LIN {X 0,Y 144.549,Z 370.18,A -85,B 0,C 180,E1 -24511.717,E2 -24511.717} C_VEL
LIN {X 0,Y 147,Z 373.251,A -85,B 0,C 180,E1 -24513.717,E2 -24513.717} C_VEL
LIN {X 0,Y 149.193,Z 377.596,A -85,B 0,C 180,E1 -24515.66,E2 -24515.66} C_VEL
LIN {X 0,Y 150.4,Z 379.371,A -85,B 0,C 180,E1 -24516.571,E2 -24516.571} C_VEL
LIN {X 0,Y 153.159,Z 385.359,A -85,B 0,C 180,E1 -24519.038,E2 -24519.038} C_VEL
LIN {X 0,Y 155.845,Z 391.898,A -85,B 0,C 180,E1 -24521.494,E2 -24521.494} C_VEL
LIN {X 0,Y 158.018,Z 400.093,A -85,B 0,C 180,E1 -24524.224,E2 -24524.224} C_VEL
LIN {X 0,Y 159.382,Z 409.972,A -85,B 0,C 180,E1 -24527.295,E2 -24527.295} C_VEL
LIN {X 0,Y 159.68,Z 420.278,A -85,B 0,C 180,E1 -24530.574,E2 -24530.574} C_VEL
LIN {X 0,Y 159.24,Z 428.16,A -85,B 0,C 180,E1 -24533.244,E2 -24533.244} C_VEL
LIN {X 0,Y 158.452,Z 434.433,A -85,B 0,C 180,E1 -24535.562,E2 -24535.562} C_VEL
LIN {X 0,Y 157.349,Z 437.828,A -85,B 0,C 180,E1 -24536.829,E2 -24536.829} C_VEL
LIN {X 0,Y 154.356,Z 444.029,A -85,B 0,C 180,E1 -24539.188,E2 -24539.188} C_VEL
LIN {X 0,Y 151.022,Z 450.566,A -85,B 0,C 180,E1 -24542.266,E2 -24542.266} C_VEL
LIN {X 0,Y 148.76,Z 455.072,A -85,B 0,C 180,E1 -24544.837,E2 -24544.837} C_VEL
LIN {X 0,Y 145.707,Z 460.563,A -85,B 0,C 180,E1 -24548.792,E2 -24548.792} C_VEL
LIN {X 0,Y 143.312,Z 464.89,A -85,B 0,C 180,E1 -24552.888,E2 -24552.888} C_VEL
LIN {X 0,Y 142.247,Z 467.263,A -85,B 0,C 180,E1 -24555.698,E2 -24555.698} C_VEL
LIN {X 0,Y 141.417,Z 469.068,A -85,B 0,C 180,E1 -24558.534,E2 -24558.534} C_VEL
LIN {X 0,Y 140.617,Z 471.529,A -85,B 0,C 180,E1 -24564.263,E2 -24564.263} C_VEL
LIN {X 0,Y 140.572,Z 472.282,A -85,B 0,C 180,E1 -24569.356,E2 -24569.356} C_VEL
LIN {X 0,Y 140.49,Z 472.123,A -85,B 0,C 180,E1 -24572.867,E2 -24572.867} C_VEL
LIN {X 0,Y 140.558,Z 471.527,A -85,B 0,C 180,E1 -24575.739,E2 -24575.739} C_VEL
LIN {X 0,Y 141.417,Z 469.068,A -85,B 0,C 180,E1 -24581.466,E2 -24581.466} C_VEL
LIN {X 0,Y 142.743,Z 466.11,A -85,B 0,C 180,E1 -24585.712,E2 -24585.712} C_VEL
LIN {X 0,Y 144.851,Z 462.118,A -85,B 0,C 180,E1 -24589.854,E2 -24589.854} C_VEL
LIN {X 0,Y 147.632,Z 456.986,A -85,B 0,C 180,E1 -24593.869,E2 -24593.869} C_VEL
LIN {X 0,Y 150.506,Z 451.725,A -85,B 0,C 180,E1 -24597.083,E2 -24597.083} C_VEL
LIN {X 0,Y 153.633,Z 445.404,A -85,B 0,C 180,E1 -24600.212,E2 -24600.212} C_VEL
LIN {X 0,Y 156.52,Z 439.453,A -85,B 0,C 180,E1 -24602.603,E2 -24602.603} C_VEL
LIN {X 0,Y 158.012,Z 436.197,A -85,B 0,C 180,E1 -24603.777,E2 -24603.777} C_VEL
LIN {X 0,Y 159.052,Z 429.716,A -85,B 0,C 180,E1 -24606.175,E2 -24606.175} C_VEL
LIN {X 0,Y 159.597,Z 422.251,A -85,B 0,C 180,E1 -24608.752,E2 -24608.752} C_VEL
LIN {X 0,Y 159.582,Z 414.231,A -85,B 0,C 180,E1 -24611.345,E2 -24611.345} C_VEL
LIN {X 0,Y 158.977,Z 406.419,A -85,B 0,C 180,E1 -24613.776,E2 -24613.776} C_VEL
LIN {X 0,Y 157.376,Z 397.352,A -85,B 0,C 180,E1 -24616.635,E2 -24616.635} C_VEL
LIN {X 0,Y 154.927,Z 389.38,A -85,B 0,C 180,E1 -24619.399,E2 -24619.399} C_VEL
LIN {X 0,Y 152.629,Z 383.818,A -85,B 0,C 180,E1 -24621.516,E2 -24621.516} C_VEL
LIN {X 0,Y 150.401,Z 379.369,A -85,B 0,C 180,E1 -24623.429,E2 -24623.429} C_VEL
LIN {X 0,Y 147.643,Z 374.742,A -85,B 0,C 180,E1 -24625.66,E2 -24625.66} C_VEL
LIN {X 0,Y 147.013,Z 373.191,A -85,B 0,C 180,E1 -24626.286,E2 -24626.286} C_VEL
LIN {X 0,Y 144.636,Z 370.361,A -85,B 0,C 180,E1 -24628.202,E2 -24628.202} C_VEL
LIN {X 0,Y 143.643,Z 367.692,A -85,B 0,C 180,E1 -24629.188,E2 -24629.188} C_VEL
LIN {X 0,Y 143.541,Z 367.179,A -85,B 0,C 180,E1 -24629.469,E2 -24629.469} C_VEL
LIN {X 0,Y 143.504,Z 367.059,A -85,B 0,C 180,E1 -24629.933,E2 -24629.933} C_VEL
LIN {X 0,Y 142.747,Z 366.562,A -85,B 0,C 180,E1 -24632.267,E2 -24632.267} C_VEL
LIN {X 0,Y 141.148,Z 366.234,A -85,B 0,C 180,E1 -24634.575,E2 -24634.575} C_VEL
LIN {X 0,Y 136.612,Z 365.578,A -85,B 0,C 180,E1 -24640.934,E2 -24640.934} C_VEL
LIN {X 0,Y 136.249,Z 365.35,A -85,B 0,C 180,E1 -24642.612,E2 -24642.612} C_VEL
LIN {X 0,Y 136.498,Z 364.983,A -85,B 0,C 180,E1 -24648.113,E2 -24648.113} C_VEL
LIN {X 0,Y 136.59,Z 364.972,A -85,B 0,C 180,E1 -24651.119,E2 -24651.119} C_VEL
LIN {X 0,Y 137.133,Z 364.867,A -85,B 0,C 180,E1 -24659.998,E2 -24659.998} C_VEL
LIN {X 0,Y 136.588,Z 364.962,A -85,B 0,C 180,E1 -24668.878,E2 -24668.878} C_VEL
LIN {X 0,Y 136.491,Z 364.984,A -85,B 0,C 180,E1 -24671.953,E2 -24671.953} C_VEL
LIN {X 0,Y 136.243,Z 365.011,A -85,B 0,C 180,E1 -24678.028,E2 -24678.028} C_VEL
LIN {X 0,Y 136.195,Z 365.018,A -85,B 0,C 180,E1 -24681.745,E2 -24681.745} C_VEL
LIN {X 0,Y 136.072,Z 365.05,A -85,B 0,C 180,E1 -24685.117,E2 -24685.117} C_VEL
LIN {X 0,Y 136.885,Z 367.482,A -85,B 0,C 180,E1 -24686.283,E2 -24686.283} C_VEL
LIN {X 0,Y 139.006,Z 369.899,A -85,B 0,C 180,E1 -24688.562,E2 -24688.562} C_VEL
LIN {X 0,Y 140.078,Z 370.732,A -85,B 0,C 180,E1 -24689.546,E2 -24689.546} C_VEL
LIN {X 0,Y 141.571,Z 373.697,A -85,B 0,C 180,E1 -24691.206,E2 -24691.206} C_VEL
LIN {X 0,Y 143.657,Z 376.017,A -85,B 0,C 180,E1 -24693.014,E2 -24693.014} C_VEL
LIN {X 0,Y 145.288,Z 378.918,A -85,B 0,C 180,E1 -24694.681,E2 -24694.681} C_VEL
LIN {X 0,Y 146.643,Z 381.055,A -85,B 0,C 180,E1 -24695.949,E2 -24695.949} C_VEL
LIN {X 0,Y 150.21,Z 387.174,A -85,B 0,C 180,E1 -24699.196,E2 -24699.196} C_VEL
LIN {X 0,Y 154.208,Z 395.585,A -85,B 0,C 180,E1 -24703.125,E2 -24703.125} C_VEL
LIN {X 0,Y 157.583,Z 404.814,A -85,B 0,C 180,E1 -24707.071,E2 -24707.071} C_VEL
LIN {X 0,Y 159.742,Z 412.862,A -85,B 0,C 180,E1 -24710.371,E2 -24710.371} C_VEL
LIN {X 0,Y 161.215,Z 420.7,A -85,B 0,C 180,E1 -24713.626,E2 -24713.626} C_VEL
LIN {X 0,Y 162.339,Z 429.067,A -85,B 0,C 180,E1 -24717.358,E2 -24717.358} C_VEL
LIN {X 0,Y 164.398,Z 436.642,A -85,B 0,C 180,E1 -24721.38,E2 -24721.38} C_VEL
LIN {X 0,Y 167.404,Z 442.696,A -85,B 0,C 180,E1 -24725.177,E2 -24725.177} C_VEL
LIN {X 0,Y 172.404,Z 448.692,A -85,B 0,C 180,E1 -24729.647,E2 -24729.647} C_VEL
LIN {X 0,Y 176.708,Z 452.183,A -85,B 0,C 180,E1 -24732.65,E2 -24732.65} C_VEL
LIN {X 0,Y 183.948,Z 456.194,A -85,B 0,C 180,E1 -24736.748,E2 -24736.748} C_VEL
LIN {X 0,Y 192.327,Z 459.212,A -85,B 0,C 180,E1 -24740.613,E2 -24740.613} C_VEL
LIN {X 0,Y 200.809,Z 461.137,A -85,B 0,C 180,E1 -24743.973,E2 -24743.973} C_VEL
LIN {X 0,Y 206.606,Z 462.007,A -85,B 0,C 180,E1 -24746.099,E2 -24746.099} C_VEL
LIN {X 0,Y 211.968,Z 462.427,A -85,B 0,C 180,E1 -24748.1,E2 -24748.1} C_VEL
LIN {X 0,Y 216.26,Z 462.479,A -85,B 0,C 180,E1 -24750,E2 -24750} C_VEL
LIN {X 0,Y 211.001,Z 462.357,A -85,B 0,C 180,E1 -24752.268,E2 -24752.268} C_VEL
LIN {X 0,Y 204.488,Z 461.751,A -85,B 0,C 180,E1 -24754.674,E2 -24754.674} C_VEL
LIN {X 0,Y 195.012,Z 459.95,A -85,B 0,C 180,E1 -24758.288,E2 -24758.288} C_VEL
LIN {X 0,Y 186.73,Z 457.364,A -85,B 0,C 180,E1 -24761.89,E2 -24761.89} C_VEL
LIN {X 0,Y 178.969,Z 453.628,A -85,B 0,C 180,E1 -24765.955,E2 -24765.955} C_VEL
LIN {X 0,Y 174.544,Z 450.62,A -85,B 0,C 180,E1 -24768.791,E2 -24768.791} C_VEL
LIN {X 0,Y 169.212,Z 445.25,A -85,B 0,C 180,E1 -24773.038,E2 -24773.038} C_VEL
LIN {X 0,Y 165.598,Z 439.388,A -85,B 0,C 180,E1 -24776.974,E2 -24776.974} C_VEL
LIN {X 0,Y 163.29,Z 433.068,A -85,B 0,C 180,E1 -24780.596,E2 -24780.596} C_VEL
LIN {X 0,Y 161.752,Z 425.235,A -85,B 0,C 180,E1 -24784.391,E2 -24784.391} C_VEL
LIN {X 0,Y 160.923,Z 418.763,A -85,B 0,C 180,E1 -24787.157,E2 -24787.157} C_VEL
LIN {X 0,Y 159.111,Z 410.213,A -85,B 0,C 180,E1 -24790.681,E2 -24790.681} C_VEL
LIN {X 0,Y 156.632,Z 401.905,A -85,B 0,C 180,E1 -24794.12,E2 -24794.12} C_VEL
LIN {X 0,Y 152.879,Z 392.58,A -85,B 0,C 180,E1 -24798.199,E2 -24798.199} C_VEL
LIN {X 0,Y 148.813,Z 384.555,A -85,B 0,C 180,E1 -24802.126,E2 -24802.126} C_VEL
LIN {X 0,Y 145.995,Z 379.751,A -85,B 0,C 180,E1 -24804.716,E2 -24804.716} C_VEL
LIN {X 0,Y 143.91,Z 376.585,A -85,B 0,C 180,E1 -24806.707,E2 -24806.707} C_VEL
LIN {X 0,Y 143.077,Z 375.23,A -85,B 0,C 180,E1 -24807.505,E2 -24807.505} C_VEL
LIN {X 0,Y 140.821,Z 372.533,A -85,B 0,C 180,E1 -24809.546,E2 -24809.546} C_VEL
LIN {X 0,Y 139.937,Z 370.486,A -85,B 0,C 180,E1 -24810.609,E2 -24810.609} C_VEL
LIN {X 0,Y 137.39,Z 368.266,A -85,B 0,C 180,E1 -24813.105,E2 -24813.105} C_VEL
LIN {X 0,Y 136.236,Z 365.864,A -85,B 0,C 180,E1 -24814.609,E2 -24814.609} C_VEL
LIN {X 0,Y 136.075,Z 365.024,A -85,B 0,C 180,E1 -24814.986,E2 -24814.986} C_VEL
LIN {X 0,Y 136.24,Z 365.008,A -85,B 0,C 180,E1 -24818.834,E2 -24818.834} C_VEL
LIN {X 0,Y 136.275,Z 365,A -85,B 0,C 180,E1 -24825.059,E2 -24825.059} C_VEL
LIN {X 0,Y 136.497,Z 364.983,A -85,B 0,C 180,E1 -24828.116,E2 -24828.116} C_VEL
LIN {X 0,Y 136.588,Z 364.962,A -85,B 0,C 180,E1 -24831.122,E2 -24831.122} C_VEL
LIN {X 0,Y 137.133,Z 364.867,A -85,B 0,C 180,E1 -24840.002,E2 -24840.002} C_VEL
LIN {X 0,Y 136.59,Z 364.971,A -85,B 0,C 180,E1 -24848.881,E2 -24848.881} C_VEL
LIN {X 0,Y 136.492,Z 364.987,A -85,B 0,C 180,E1 -24851.956,E2 -24851.956} C_VEL
LIN {X 0,Y 136.266,Z 365.014,A -85,B 0,C 180,E1 -24854.946,E2 -24854.946} C_VEL
LIN {X 0,Y 136.365,Z 366.025,A -85,B 0,C 180,E1 -24861.149,E2 -24861.149} C_VEL
LIN {X 0,Y 136.373,Z 366.981,A -85,B 0,C 180,E1 -24865.163,E2 -24865.163} C_VEL
LIN {X 0,Y 137.366,Z 369.881,A -85,B 0,C 180,E1 -24866.494,E2 -24866.494} C_VEL
LIN {X 0,Y 139.889,Z 372.994,A -85,B 0,C 180,E1 -24869.09,E2 -24869.09} C_VEL
LIN {X 0,Y 140.452,Z 373.735,A -85,B 0,C 180,E1 -24869.645,E2 -24869.645} C_VEL
LIN {X 0,Y 141.954,Z 377.052,A -85,B 0,C 180,E1 -24871.324,E2 -24871.324} C_VEL
LIN {X 0,Y 143.821,Z 379.604,A -85,B 0,C 180,E1 -24872.975,E2 -24872.975} C_VEL
LIN {X 0,Y 144.834,Z 382.056,A -85,B 0,C 180,E1 -24874.089,E2 -24874.089} C_VEL
LIN {X 0,Y 146.097,Z 384.055,A -85,B 0,C 180,E1 -24875.26,E2 -24875.26} C_VEL
LIN {X 0,Y 149.265,Z 391.3,A -85,B 0,C 180,E1 -24878.473,E2 -24878.473} C_VEL
LIN {X 0,Y 151.684,Z 399.019,A -85,B 0,C 180,E1 -24881.508,E2 -24881.508} C_VEL
LIN {X 0,Y 152.964,Z 406.059,A -85,B 0,C 180,E1 -24883.989,E2 -24883.989} C_VEL
LIN {X 0,Y 153.587,Z 414.007,A -85,B 0,C 180,E1 -24886.656,E2 -24886.656} C_VEL
LIN {X 0,Y 153.528,Z 422.357,A -85,B 0,C 180,E1 -24889.526,E2 -24889.526} C_VEL
LIN {X 0,Y 152.845,Z 430.118,A -85,B 0,C 180,E1 -24892.368,E2 -24892.368} C_VEL
LIN {X 0,Y 151.94,Z 435.994,A -85,B 0,C 180,E1 -24894.677,E2 -24894.677} C_VEL
LIN {X 0,Y 150.614,Z 439.258,A -85,B 0,C 180,E1 -24895.948,E2 -24895.948} C_VEL
LIN {X 0,Y 147.524,Z 445.208,A -85,B 0,C 180,E1 -24898.397,E2 -24898.397} C_VEL
LIN {X 0,Y 144.204,Z 451.389,A -85,B 0,C 180,E1 -24901.535,E2 -24901.535} C_VEL
LIN {X 0,Y 142.365,Z 454.876,A -85,B 0,C 180,E1 -24903.622,E2 -24903.622} C_VEL
LIN {X 0,Y 139.085,Z 460.367,A -85,B 0,C 180,E1 -24907.73,E2 -24907.73} C_VEL
LIN {X 0,Y 136.507,Z 464.693,A -85,B 0,C 180,E1 -24912.007,E2 -24912.007} C_VEL
LIN {X 0,Y 135.35,Z 467.067,A -85,B 0,C 180,E1 -24914.952,E2 -24914.952} C_VEL
LIN {X 0,Y 134.451,Z 468.872,A -85,B 0,C 180,E1 -24917.931,E2 -24917.931} C_VEL
LIN {X 0,Y 133.543,Z 471.333,A -85,B 0,C 180,E1 -24923.958,E2 -24923.958} C_VEL
LIN {X 0,Y 133.414,Z 471.927,A -85,B 0,C 180,E1 -24926.98,E2 -24926.98} C_VEL
LIN {X 0,Y 133.535,Z 472.088,A -85,B 0,C 180,E1 -24930,E2 -24930} C_VEL
LIN {X 0,Y 133.401,Z 471.927,A -85,B 0,C 180,E1 -24933.02,E2 -24933.02} C_VEL
LIN {X 0,Y 133.474,Z 471.331,A -85,B 0,C 180,E1 -24936.045,E2 -24936.045} C_VEL
LIN {X 0,Y 134.451,Z 468.872,A -85,B 0,C 180,E1 -24942.069,E2 -24942.069} C_VEL
LIN {X 0,Y 135.882,Z 465.913,A -85,B 0,C 180,E1 -24946.527,E2 -24946.527} C_VEL
LIN {X 0,Y 138.157,Z 461.921,A -85,B 0,C 180,E1 -24950.86,E2 -24950.86} C_VEL
LIN {X 0,Y 141.146,Z 456.79,A -85,B 0,C 180,E1 -24955.039,E2 -24955.039} C_VEL
LIN {X 0,Y 143.579,Z 452.685,A -85,B 0,C 180,E1 -24957.711,E2 -24957.711} C_VEL
LIN {X 0,Y 146.722,Z 446.721,A -85,B 0,C 180,E1 -24960.912,E2 -24960.912} C_VEL
LIN {X 0,Y 149.771,Z 440.883,A -85,B 0,C 180,E1 -24963.461,E2 -24963.461} C_VEL
LIN {X 0,Y 151.95,Z 435.994,A -85,B 0,C 180,E1 -24965.32,E2 -24965.32} C_VEL
LIN {X 0,Y 153.22,Z 427.209,A -85,B 0,C 180,E1 -24968.759,E2 -24968.759} C_VEL
LIN {X 0,Y 153.66,Z 417.036,A -85,B 0,C 180,E1 -24972.333,E2 -24972.333} C_VEL
LIN {X 0,Y 153.18,Z 408.386,A -85,B 0,C 180,E1 -24975.269,E2 -24975.269} C_VEL
LIN {X 0,Y 152.083,Z 400.634,A -85,B 0,C 180,E1 -24977.924,E2 -24977.924} C_VEL
LIN {X 0,Y 149.973,Z 393.209,A -85,B 0,C 180,E1 -24980.705,E2 -24980.705} C_VEL
LIN {X 0,Y 147.368,Z 387.012,A -85,B 0,C 180,E1 -24983.405,E2 -24983.405} C_VEL
LIN {X 0,Y 145.745,Z 383.501,A -85,B 0,C 180,E1 -24985.06,E2 -24985.06} C_VEL
LIN {X 0,Y 143.906,Z 379.83,A -85,B 0,C 180,E1 -24986.932,E2 -24986.932} C_VEL
LIN {X 0,Y 143.251,Z 378.671,A -85,B 0,C 180,E1 -24987.546,E2 -24987.546} C_VEL
LIN {X 0,Y 141.051,Z 375.424,A -85,B 0,C 180,E1 -24989.598,E2 -24989.598} C_VEL
LIN {X 0,Y 140.309,Z 373.275,A -85,B 0,C 180,E1 -24990.551,E2 -24990.551} C_VEL
LIN {X 0,Y 137.672,Z 370.389,A -85,B 0,C 180,E1 -24993.161,E2 -24993.161} C_VEL
LIN {X 0,Y 136.526,Z 367.751,A -85,B 0,C 180,E1 -24994.562,E2 -24994.562} C_VEL
LIN {X 0,Y 136.352,Z 366.837,A -85,B 0,C 180,E1 -24995.037,E2 -24995.037} C_VEL
LIN {X 0,Y 136.365,Z 366.023,A -85,B 0,C 180,E1 -24998.851,E2 -24998.851} C_VEL
LIN {X 0,Y 136.249,Z 365.35,A -85,B 0,C 180,E1 -25002.612,E2 -25002.612} C_VEL
LIN {X 0,Y 135.519,Z 365.197,A -85,B 0,C 180,E1 -25005.082,E2 -25005.082} C_VEL
LIN {X 0,Y 133.954,Z 365.311,A -85,B 0,C 180,E1 -25007.524,E2 -25007.524} C_VEL
LIN {X 0,Y 129.763,Z 365.821,A -85,B 0,C 180,E1 -25014.266,E2 -25014.266} C_VEL
LIN {X 0,Y 129.594,Z 365.838,A -85,B 0,C 180,E1 -25016.037,E2 -25016.037} C_VEL
LIN {X 0,Y 130.089,Z 365.742,A -85,B 0,C 180,E1 -25019.998,E2 -25019.998} C_VEL
LIN {X 0,Y 129.514,Z 365.841,A -85,B 0,C 180,E1 -25029.367,E2 -25029.367} C_VEL
LIN {X 0,Y 129.392,Z 365.867,A -85,B 0,C 180,E1 -25032.546,E2 -25032.546} C_VEL
LIN {X 0,Y 129.195,Z 365.966,A -85,B 0,C 180,E1 -25037.611,E2 -25037.611} C_VEL
LIN {X 0,Y 129.963,Z 368.398,A -85,B 0,C 180,E1 -25039.341,E2 -25039.341} C_VEL
LIN {X 0,Y 132.558,Z 371.16,A -85,B 0,C 180,E1 -25043.164,E2 -25043.164} C_VEL
LIN {X 0,Y 133.403,Z 371.849,A -85,B 0,C 180,E1 -25044.199,E2 -25044.199} C_VEL
LIN {X 0,Y 134.71,Z 374.594,A -85,B 0,C 180,E1 -25046.114,E2 -25046.114} C_VEL
LIN {X 0,Y 137.334,Z 377.785,A -85,B 0,C 180,E1 -25049.088,E2 -25049.088} C_VEL
LIN {X 0,Y 138.437,Z 379.851,A -85,B 0,C 180,E1 -25050.507,E2 -25050.507} C_VEL
LIN {X 0,Y 139.789,Z 381.355,A -85,B 0,C 180,E1 -25051.861,E2 -25051.861} C_VEL
LIN {X 0,Y 142.96,Z 387.002,A -85,B 0,C 180,E1 -25055.329,E2 -25055.329} C_VEL
LIN {X 0,Y 146.054,Z 392.9,A -85,B 0,C 180,E1 -25058.72,E2 -25058.72} C_VEL
LIN {X 0,Y 148.85,Z 399.387,A -85,B 0,C 180,E1 -25062.015,E2 -25062.015} C_VEL
LIN {X 0,Y 151.26,Z 406.1,A -85,B 0,C 180,E1 -25065.172,E2 -25065.172} C_VEL
LIN {X 0,Y 153.417,Z 414.339,A -85,B 0,C 180,E1 -25068.875,E2 -25068.875} C_VEL
LIN {X 0,Y 154.742,Z 421.474,A -85,B 0,C 180,E1 -25072.076,E2 -25072.076} C_VEL
LIN {X 0,Y 155.583,Z 429.848,A -85,B 0,C 180,E1 -25076.024,E2 -25076.024} C_VEL
LIN {X 0,Y 157.092,Z 436.938,A -85,B 0,C 180,E1 -25079.952,E2 -25079.952} C_VEL
LIN {X 0,Y 159.45,Z 442.933,A -85,B 0,C 180,E1 -25083.848,E2 -25083.848} C_VEL
LIN {X 0,Y 162.32,Z 447.239,A -85,B 0,C 180,E1 -25087.066,E2 -25087.066} C_VEL
LIN {X 0,Y 167.761,Z 452.382,A -85,B 0,C 180,E1 -25091.646,E2 -25091.646} C_VEL
LIN {X 0,Y 174.643,Z 456.453,A -85,B 0,C 180,E1 -25096.028,E2 -25096.028} C_VEL
LIN {X 0,Y 179.807,Z 458.597,A -85,B 0,C 180,E1 -25098.73,E2 -25098.73} C_VEL
LIN {X 0,Y 185.351,Z 460.215,A -85,B 0,C 180,E1 -25101.276,E2 -25101.276} C_VEL
LIN {X 0,Y 197.268,Z 462.281,A -85,B 0,C 180,E1 -25105.967,E2 -25105.967} C_VEL
LIN {X 0,Y 203.889,Z 462.736,A -85,B 0,C 180,E1 -25108.383,E2 -25108.383} C_VEL
LIN {X 0,Y 207.904,Z 462.705,A -85,B 0,C 180,E1 -25110,E2 -25110} C_VEL
LIN {X 0,Y 202.898,Z 462.676,A -85,B 0,C 180,E1 -25111.985,E2 -25111.985} C_VEL
LIN {X 0,Y 197.114,Z 462.268,A -85,B 0,C 180,E1 -25114.089,E2 -25114.089} C_VEL
LIN {X 0,Y 184.948,Z 460.105,A -85,B 0,C 180,E1 -25118.894,E2 -25118.894} C_VEL
LIN {X 0,Y 179.301,Z 458.436,A -85,B 0,C 180,E1 -25121.51,E2 -25121.51} C_VEL
LIN {X 0,Y 172.165,Z 455.285,A -85,B 0,C 180,E1 -25125.4,E2 -25125.4} C_VEL
LIN {X 0,Y 165.041,Z 450.088,A -85,B 0,C 180,E1 -25130.478,E2 -25130.478} C_VEL
LIN {X 0,Y 160.648,Z 444.842,A -85,B 0,C 180,E1 -25134.747,E2 -25134.747} C_VEL
LIN {X 0,Y 157.742,Z 438.97,A -85,B 0,C 180,E1 -25138.792,E2 -25138.792} C_VEL
LIN {X 0,Y 155.948,Z 432.198,A -85,B 0,C 180,E1 -25142.738,E2 -25142.738} C_VEL
LIN {X 0,Y 155.14,Z 425.458,A -85,B 0,C 180,E1 -25146.08,E2 -25146.08} C_VEL
LIN {X 0,Y 154.234,Z 418.559,A -85,B 0,C 180,E1 -25149.23,E2 -25149.23} C_VEL
LIN {X 0,Y 152.654,Z 411.161,A -85,B 0,C 180,E1 -25152.558,E2 -25152.558} C_VEL
LIN {X 0,Y 150.058,Z 402.564,A -85,B 0,C 180,E1 -25156.485,E2 -25156.485} C_VEL
LIN {X 0,Y 146.805,Z 394.481,A -85,B 0,C 180,E1 -25160.474,E2 -25160.474} C_VEL
LIN {X 0,Y 142.219,Z 385.404,A -85,B 0,C 180,E1 -25165.553,E2 -25165.553} C_VEL
LIN {X 0,Y 139.791,Z 381.35,A -85,B 0,C 180,E1 -25168.139,E2 -25168.139} C_VEL
LIN {X 0,Y 138.074,Z 379.289,A -85,B 0,C 180,E1 -25169.917,E2 -25169.917} C_VEL
LIN {X 0,Y 136.128,Z 376.132,A -85,B 0,C 180,E1 -25172.314,E2 -25172.314} C_VEL
LIN {X 0,Y 134.032,Z 373.451,A -85,B 0,C 180,E1 -25174.786,E2 -25174.786} C_VEL
LIN {X 0,Y 133.219,Z 371.497,A -85,B 0,C 180,E1 -25176.076,E2 -25176.076} C_VEL
LIN {X 0,Y 130.785,Z 369.58,A -85,B 0,C 180,E1 -25179.26,E2 -25179.26} C_VEL
LIN {X 0,Y 129.508,Z 367.278,A -85,B 0,C 180,E1 -25181.615,E2 -25181.615} C_VEL
LIN {X 0,Y 129.198,Z 365.892,A -85,B 0,C 180,E1 -25182.593,E2 -25182.593} C_VEL
LIN {X 0,Y 129.416,Z 365.865,A -85,B 0,C 180,E1 -25187.822,E2 -25187.822} C_VEL
LIN {X 0,Y 129.514,Z 365.841,A -85,B 0,C 180,E1 -25190.633,E2 -25190.633} C_VEL
LIN {X 0,Y 130.089,Z 365.742,A -85,B 0,C 180,E1 -25200.002,E2 -25200.002} C_VEL
LIN {X 0,Y 129.516,Z 365.853,A -85,B 0,C 180,E1 -25209.371,E2 -25209.371} C_VEL
LIN {X 0,Y 129.393,Z 365.87,A -85,B 0,C 180,E1 -25212.55,E2 -25212.55} C_VEL
LIN {X 0,Y 129.26,Z 366.565,A -85,B 0,C 180,E1 -25217.3,E2 -25217.3} C_VEL
LIN {X 0,Y 130.364,Z 369.612,A -85,B 0,C 180,E1 -25219.487,E2 -25219.487} C_VEL
LIN {X 0,Y 133.365,Z 373.074,A -85,B 0,C 180,E1 -25223.694,E2 -25223.694} C_VEL
LIN {X 0,Y 134.064,Z 374.821,A -85,B 0,C 180,E1 -25224.797,E2 -25224.797} C_VEL
LIN {X 0,Y 135.889,Z 377.961,A -85,B 0,C 180,E1 -25227.116,E2 -25227.116} C_VEL
LIN {X 0,Y 137.262,Z 379.724,A -85,B 0,C 180,E1 -25228.583,E2 -25228.583} C_VEL
LIN {X 0,Y 138.775,Z 383.146,A -85,B 0,C 180,E1 -25230.579,E2 -25230.579} C_VEL
LIN {X 0,Y 139.952,Z 384.871,A -85,B 0,C 180,E1 -25231.822,E2 -25231.822} C_VEL
LIN {X 0,Y 143.488,Z 392.866,A -85,B 0,C 180,E1 -25236,E2 -25236} C_VEL
LIN {X 0,Y 145.644,Z 399.158,A -85,B 0,C 180,E1 -25238.854,E2 -25238.854} C_VEL
LIN {X 0,Y 147.188,Z 406.936,A -85,B 0,C 180,E1 -25241.952,E2 -25241.952} C_VEL
LIN {X 0,Y 147.76,Z 415.669,A -85,B 0,C 180,E1 -25245.148,E2 -25245.148} C_VEL
LIN {X 0,Y 147.446,Z 423.791,A -85,B 0,C 180,E1 -25248.14,E2 -25248.14} C_VEL
LIN {X 0,Y 146.822,Z 430.078,A -85,B 0,C 180,E1 -25250.611,E2 -25250.611} C_VEL
LIN {X 0,Y 145.846,Z 435.786,A -85,B 0,C 180,E1 -25252.962,E2 -25252.962} C_VEL
LIN {X 0,Y 144.754,Z 439.061,A -85,B 0,C 180,E1 -25254.365,E2 -25254.365} C_VEL
LIN {X 0,Y 141.5,Z 445.011,A -85,B 0,C 180,E1 -25256.883,E2 -25256.883} C_VEL
LIN {X 0,Y 137.66,Z 451.732,A -85,B 0,C 180,E1 -25260.44,E2 -25260.44} C_VEL
LIN {X 0,Y 134.729,Z 456.593,A -85,B 0,C 180,E1 -25263.68,E2 -25263.68} C_VEL
LIN {X 0,Y 131.515,Z 461.724,A -85,B 0,C 180,E1 -25268.033,E2 -25268.033} C_VEL
LIN {X 0,Y 129.059,Z 465.716,A -85,B 0,C 180,E1 -25272.572,E2 -25272.572} C_VEL
LIN {X 0,Y 127.48,Z 468.675,A -85,B 0,C 180,E1 -25277.26,E2 -25277.26} C_VEL
LIN {X 0,Y 126.464,Z 471.136,A -85,B 0,C 180,E1 -25283.619,E2 -25283.619} C_VEL
LIN {X 0,Y 126.317,Z 471.731,A -85,B 0,C 180,E1 -25286.811,E2 -25286.811} C_VEL
LIN {X 0,Y 126.431,Z 471.892,A -85,B 0,C 180,E1 -25290,E2 -25290} C_VEL
LIN {X 0,Y 126.306,Z 471.731,A -85,B 0,C 180,E1 -25293.19,E2 -25293.19} C_VEL
LIN {X 0,Y 126.415,Z 471.135,A -85,B 0,C 180,E1 -25296.384,E2 -25296.384} C_VEL
LIN {X 0,Y 127.48,Z 468.675,A -85,B 0,C 180,E1 -25302.74,E2 -25302.74} C_VEL
LIN {X 0,Y 129.059,Z 465.716,A -85,B 0,C 180,E1 -25307.428,E2 -25307.428} C_VEL
LIN {X 0,Y 131.517,Z 461.724,A -85,B 0,C 180,E1 -25311.967,E2 -25311.967} C_VEL
LIN {X 0,Y 134.732,Z 456.593,A -85,B 0,C 180,E1 -25316.32,E2 -25316.32} C_VEL
LIN {X 0,Y 137.786,Z 451.564,A -85,B 0,C 180,E1 -25319.652,E2 -25319.652} C_VEL
LIN {X 0,Y 141.47,Z 445.01,A -85,B 0,C 180,E1 -25323.124,E2 -25323.124} C_VEL
LIN {X 0,Y 144.726,Z 439.06,A -85,B 0,C 180,E1 -25325.643,E2 -25325.643} C_VEL
LIN {X 0,Y 145.449,Z 437.429,A -85,B 0,C 180,E1 -25326.293,E2 -25326.293} C_VEL
LIN {X 0,Y 146.81,Z 430.038,A -85,B 0,C 180,E1 -25329.411,E2 -25329.411} C_VEL
LIN {X 0,Y 147.557,Z 422.469,A -85,B 0,C 180,E1 -25332.349,E2 -25332.349} C_VEL
LIN {X 0,Y 147.725,Z 414.673,A -85,B 0,C 180,E1 -25335.215,E2 -25335.215} C_VEL
LIN {X 0,Y 147.15,Z 407.03,A -85,B 0,C 180,E1 -25338.035,E2 -25338.035} C_VEL
LIN {X 0,Y 145.923,Z 400.209,A -85,B 0,C 180,E1 -25340.725,E2 -25340.725} C_VEL
LIN {X 0,Y 143.485,Z 392.874,A -85,B 0,C 180,E1 -25343.999,E2 -25343.999} C_VEL
LIN {X 0,Y 141.079,Z 387.623,A -85,B 0,C 180,E1 -25346.77,E2 -25346.77} C_VEL
LIN {X 0,Y 139.952,Z 384.873,A -85,B 0,C 180,E1 -25348.178,E2 -25348.178} C_VEL
LIN {X 0,Y 138.093,Z 381.872,A -85,B 0,C 180,E1 -25350.249,E2 -25350.249} C_VEL
LIN {X 0,Y 136.883,Z 379.061,A -85,B 0,C 180,E1 -25351.852,E2 -25351.852} C_VEL
LIN {X 0,Y 134.554,Z 375.996,A -85,B 0,C 180,E1 -25354.473,E2 -25354.473} C_VEL
LIN {X 0,Y 133.374,Z 373.034,A -85,B 0,C 180,E1 -25356.308,E2 -25356.308} C_VEL
LIN {X 0,Y 130.476,Z 369.806,A -85,B 0,C 180,E1 -25360.325,E2 -25360.325} C_VEL
LIN {X 0,Y 129.406,Z 367.225,A -85,B 0,C 180,E1 -25362.313,E2 -25362.313} C_VEL
LIN {X 0,Y 129.23,Z 366.43,A -85,B 0,C 180,E1 -25362.798,E2 -25362.798} C_VEL
LIN {X 0,Y 129.417,Z 365.865,A -85,B 0,C 180,E1 -25367.819,E2 -25367.819} C_VEL
LIN {X 0,Y 129.516,Z 365.852,A -85,B 0,C 180,E1 -25370.629,E2 -25370.629} C_VEL
LIN {X 0,Y 129.594,Z 365.838,A -85,B 0,C 180,E1 -25376.037,E2 -25376.037} C_VEL
LIN {X 0,Y 129.408,Z 365.958,A -85,B 0,C 180,E1 -25377.769,E2 -25377.769} C_VEL
LIN {X 0,Y 128.711,Z 366.3,A -85,B 0,C 180,E1 -25379.482,E2 -25379.482} C_VEL
LIN {X 0,Y 126.551,Z 367.451,A -85,B 0,C 180,E1 -25382.88,E2 -25382.88} C_VEL
LIN {X 0,Y 124.518,Z 368.972,A -85,B 0,C 180,E1 -25386.388,E2 -25386.388} C_VEL
LIN {X 0,Y 123.99,Z 370.153,A -85,B 0,C 180,E1 -25389.102,E2 -25389.102} C_VEL
LIN {X 0,Y 124.132,Z 370.527,A -85,B 0,C 180,E1 -25390.011,E2 -25390.011} C_VEL
LIN {X 0,Y 126.963,Z 372.862,A -85,B 0,C 180,E1 -25396.789,E2 -25396.789} C_VEL
LIN {X 0,Y 128.003,Z 375.462,A -85,B 0,C 180,E1 -25399.232,E2 -25399.232} C_VEL
LIN {X 0,Y 130.653,Z 378.237,A -85,B 0,C 180,E1 -25403.298,E2 -25403.298} C_VEL
LIN {X 0,Y 131.711,Z 380.72,A -85,B 0,C 180,E1 -25405.267,E2 -25405.267} C_VEL
LIN {X 0,Y 133.921,Z 383.641,A -85,B 0,C 180,E1 -25408.182,E2 -25408.182} C_VEL
LIN {X 0,Y 135.083,Z 385.829,A -85,B 0,C 180,E1 -25409.765,E2 -25409.765} C_VEL
LIN {X 0,Y 136.214,Z 387.222,A -85,B 0,C 180,E1 -25411.059,E2 -25411.059} C_VEL
LIN {X 0,Y 140.11,Z 394.885,A -85,B 0,C 180,E1 -25416.112,E2 -25416.112} C_VEL
LIN {X 0,Y 143.391,Z 402.735,A -85,B 0,C 180,E1 -25420.597,E2 -25420.597} C_VEL
LIN {X 0,Y 145.736,Z 410.001,A -85,B 0,C 180,E1 -25424.363,E2 -25424.363} C_VEL
LIN {X 0,Y 147.477,Z 417.732,A -85,B 0,C 180,E1 -25428.151,E2 -25428.151} C_VEL
LIN {X 0,Y 148.492,Z 424.323,A -85,B 0,C 180,E1 -25431.399,E2 -25431.399} C_VEL
LIN {X 0,Y 148.938,Z 429.995,A -85,B 0,C 180,E1 -25434.243,E2 -25434.243} C_VEL
LIN {X 0,Y 149.673,Z 436.155,A -85,B 0,C 180,E1 -25437.691,E2 -25437.691} C_VEL
LIN {X 0,Y 151.731,Z 443.17,A -85,B 0,C 180,E1 -25442.407,E2 -25442.407} C_VEL
LIN {X 0,Y 154.168,Z 447.48,A -85,B 0,C 180,E1 -25445.778,E2 -25445.778} C_VEL
LIN {X 0,Y 159.237,Z 452.828,A -85,B 0,C 180,E1 -25450.804,E2 -25450.804} C_VEL
LIN {X 0,Y 165.372,Z 456.712,A -85,B 0,C 180,E1 -25455.227,E2 -25455.227} C_VEL
LIN {X 0,Y 171.88,Z 459.349,A -85,B 0,C 180,E1 -25458.905,E2 -25458.905} C_VEL
LIN {X 0,Y 177.582,Z 460.958,A -85,B 0,C 180,E1 -25461.641,E2 -25461.641} C_VEL
LIN {X 0,Y 187.486,Z 462.532,A -85,B 0,C 180,E1 -25465.7,E2 -25465.7} C_VEL
LIN {X 0,Y 196.804,Z 463.004,A -85,B 0,C 180,E1 -25469.097,E2 -25469.097} C_VEL
LIN {X 0,Y 199.193,Z 462.941,A -85,B 0,C 180,E1 -25470,E2 -25470} C_VEL
LIN {X 0,Y 193.528,Z 462.933,A -85,B 0,C 180,E1 -25472.081,E2 -25472.081} C_VEL
LIN {X 0,Y 183.663,Z 462.021,A -85,B 0,C 180,E1 -25475.798,E2 -25475.798} C_VEL
LIN {X 0,Y 175.75,Z 460.478,A -85,B 0,C 180,E1 -25479.204,E2 -25479.204} C_VEL
LIN {X 0,Y 170.362,Z 458.863,A -85,B 0,C 180,E1 -25481.904,E2 -25481.904} C_VEL
LIN {X 0,Y 161.834,Z 454.712,A -85,B 0,C 180,E1 -25487.182,E2 -25487.182} C_VEL
LIN {X 0,Y 157.316,Z 451.118,A -85,B 0,C 180,E1 -25490.94,E2 -25490.94} C_VEL
LIN {X 0,Y 152.891,Z 445.387,A -85,B 0,C 180,E1 -25495.891,E2 -25495.891} C_VEL
LIN {X 0,Y 150.456,Z 439.525,A -85,B 0,C 180,E1 -25500.141,E2 -25500.141} C_VEL
LIN {X 0,Y 149.251,Z 433.733,A -85,B 0,C 180,E1 -25503.733,E2 -25503.733} C_VEL
LIN {X 0,Y 148.596,Z 425.684,A -85,B 0,C 180,E1 -25507.941,E2 -25507.941} C_VEL
LIN {X 0,Y 147.691,Z 418.873,A -85,B 0,C 180,E1 -25511.303,E2 -25511.303} C_VEL
LIN {X 0,Y 146.159,Z 411.717,A -85,B 0,C 180,E1 -25514.829,E2 -25514.829} C_VEL
LIN {X 0,Y 144.026,Z 404.594,A -85,B 0,C 180,E1 -25518.465,E2 -25518.465} C_VEL
LIN {X 0,Y 141.603,Z 398.337,A -85,B 0,C 180,E1 -25521.838,E2 -25521.838} C_VEL
LIN {X 0,Y 138.372,Z 391.428,A -85,B 0,C 180,E1 -25526.036,E2 -25526.036} C_VEL
LIN {X 0,Y 136.212,Z 387.227,A -85,B 0,C 180,E1 -25528.94,E2 -25528.94} C_VEL
LIN {X 0,Y 134.471,Z 384.798,A -85,B 0,C 180,E1 -25531.019,E2 -25531.019} C_VEL
LIN {X 0,Y 132.812,Z 382.052,A -85,B 0,C 180,E1 -25533.272,E2 -25533.272} C_VEL
LIN {X 0,Y 131.177,Z 379.705,A -85,B 0,C 180,E1 -25535.616,E2 -25535.616} C_VEL
LIN {X 0,Y 130.659,Z 378.218,A -85,B 0,C 180,E1 -25536.703,E2 -25536.703} C_VEL
LIN {X 0,Y 127.602,Z 374.808,A -85,B 0,C 180,E1 -25541.539,E2 -25541.539} C_VEL
LIN {X 0,Y 126.844,Z 372.589,A -85,B 0,C 180,E1 -25543.505,E2 -25543.505} C_VEL
LIN {X 0,Y 123.092,Z 367.367,A -85,B 0,C 180,E1 -25559.593,E2 -25559.593} C_VEL
LIN {X 0,Y 123.102,Z 367.357,A -85,B 0,C 180,E1 -25560.411,E2 -25560.411} C_VEL
LIN {X 0,Y 124.068,Z 370.422,A -85,B 0,C 180,E1 -25568.964,E2 -25568.964} C_VEL
LIN {X 0,Y 127.102,Z 373.253,A -85,B 0,C 180,E1 -25576.361,E2 -25576.361} C_VEL
LIN {X 0,Y 128.088,Z 376.213,A -85,B 0,C 180,E1 -25578.807,E2 -25578.807} C_VEL
LIN {X 0,Y 130.248,Z 379.018,A -85,B 0,C 180,E1 -25582.194,E2 -25582.194} C_VEL
LIN {X 0,Y 133.081,Z 384.477,A -85,B 0,C 180,E1 -25586.674,E2 -25586.674} C_VEL
LIN {X 0,Y 133.669,Z 385.217,A -85,B 0,C 180,E1 -25587.392,E2 -25587.392} C_VEL
LIN {X 0,Y 136.305,Z 390.857,A -85,B 0,C 180,E1 -25591.04,E2 -25591.04} C_VEL
LIN {X 0,Y 138.868,Z 397.41,A -85,B 0,C 180,E1 -25594.795,E2 -25594.795} C_VEL
LIN {X 0,Y 140.642,Z 403.363,A -85,B 0,C 180,E1 -25597.747,E2 -25597.747} C_VEL
LIN {X 0,Y 141.771,Z 410.205,A -85,B 0,C 180,E1 -25600.66,E2 -25600.66} C_VEL
LIN {X 0,Y 142.017,Z 418.245,A -85,B 0,C 180,E1 -25603.856,E2 -25603.856} C_VEL
LIN {X 0,Y 141.246,Z 427.588,A -85,B 0,C 180,E1 -25607.609,E2 -25607.609} C_VEL
LIN {X 0,Y 139.884,Z 435.577,A -85,B 0,C 180,E1 -25611.096,E2 -25611.096} C_VEL
LIN {X 0,Y 138.943,Z 438.862,A -85,B 0,C 180,E1 -25612.628,E2 -25612.628} C_VEL
LIN {X 0,Y 135.57,Z 444.814,A -85,B 0,C 180,E1 -25615.233,E2 -25615.233} C_VEL
LIN {X 0,Y 131.768,Z 451.026,A -85,B 0,C 180,E1 -25618.584,E2 -25618.584} C_VEL
LIN {X 0,Y 129.769,Z 454.483,A -85,B 0,C 180,E1 -25620.829,E2 -25620.829} C_VEL
LIN {X 0,Y 126.009,Z 459.974,A -85,B 0,C 180,E1 -25625.273,E2 -25625.273} C_VEL
LIN {X 0,Y 123.019,Z 464.3,A -85,B 0,C 180,E1 -25629.954,E2 -25629.954} C_VEL
LIN {X 0,Y 121.618,Z 466.673,A -85,B 0,C 180,E1 -25633.206,E2 -25633.206} C_VEL
LIN {X 0,Y 120.538,Z 468.478,A -85,B 0,C 180,E1 -25636.513,E2 -25636.513} C_VEL
LIN {X 0,Y 119.411,Z 470.94,A -85,B 0,C 180,E1 -25643.24,E2 -25643.24} C_VEL
LIN {X 0,Y 119.231,Z 471.536,A -85,B 0,C 180,E1 -25646.621,E2 -25646.621} C_VEL
LIN {X 0,Y 119.337,Z 471.696,A -85,B 0,C 180,E1 -25650,E2 -25650} C_VEL
LIN {X 0,Y 119.222,Z 471.535,A -85,B 0,C 180,E1 -25653.379,E2 -25653.379} C_VEL
LIN {X 0,Y 119.338,Z 470.938,A -85,B 0,C 180,E1 -25656.764,E2 -25656.764} C_VEL
LIN {X 0,Y 120.538,Z 468.478,A -85,B 0,C 180,E1 -25663.487,E2 -25663.487} C_VEL
LIN {X 0,Y 122.256,Z 465.519,A -85,B 0,C 180,E1 -25668.432,E2 -25668.432} C_VEL
LIN {X 0,Y 124.936,Z 461.528,A -85,B 0,C 180,E1 -25673.189,E2 -25673.189} C_VEL
LIN {X 0,Y 128.398,Z 456.397,A -85,B 0,C 180,E1 -25677.727,E2 -25677.727} C_VEL
LIN {X 0,Y 131.874,Z 450.893,A -85,B 0,C 180,E1 -25681.491,E2 -25681.491} C_VEL
LIN {X 0,Y 135.55,Z 444.814,A -85,B 0,C 180,E1 -25684.773,E2 -25684.773} C_VEL
LIN {X 0,Y 138.936,Z 438.862,A -85,B 0,C 180,E1 -25687.374,E2 -25687.374} C_VEL
LIN {X 0,Y 140.571,Z 431.863,A -85,B 0,C 180,E1 -25690.538,E2 -25690.538} C_VEL
LIN {X 0,Y 141.549,Z 424.604,A -85,B 0,C 180,E1 -25693.594,E2 -25693.594} C_VEL
LIN {X 0,Y 142.006,Z 416.978,A -85,B 0,C 180,E1 -25696.63,E2 -25696.63} C_VEL
LIN {X 0,Y 141.496,Z 407.989,A -85,B 0,C 180,E1 -25700.244,E2 -25700.244} C_VEL
LIN {X 0,Y 140.047,Z 400.993,A -85,B 0,C 180,E1 -25703.411,E2 -25703.411} C_VEL
LIN {X 0,Y 137.814,Z 394.518,A -85,B 0,C 180,E1 -25706.754,E2 -25706.754} C_VEL
LIN {X 0,Y 135.699,Z 389.661,A -85,B 0,C 180,E1 -25709.755,E2 -25709.755} C_VEL
LIN {X 0,Y 133.675,Z 385.201,A -85,B 0,C 180,E1 -25712.609,E2 -25712.609} C_VEL
LIN {X 0,Y 131.928,Z 382.742,A -85,B 0,C 180,E1 -25714.905,E2 -25714.905} C_VEL
LIN {X 0,Y 130.119,Z 378.849,A -85,B 0,C 180,E1 -25717.992,E2 -25717.992} C_VEL
LIN {X 0,Y 127.663,Z 375.325,A -85,B 0,C 180,E1 -25722.063,E2 -25722.063} C_VEL
LIN {X 0,Y 126.975,Z 372.998,A -85,B 0,C 180,E1 -25723.932,E2 -25723.932} C_VEL
LIN {X 0,Y 123.091,Z 367.382,A -85,B 0,C 180,E1 -25739.589,E2 -25739.589} C_VEL
LIN {X 0,Y 123.097,Z 367.293,A -85,B 0,C 180,E1 -25740.203,E2 -25740.203} C_VEL
LIN {X 0,Y 124.132,Z 370.527,A -85,B 0,C 180,E1 -25750.011,E2 -25750.011} C_VEL
LIN {X 0,Y 124.834,Z 372.15,A -85,B 0,C 180,E1 -25752.608,E2 -25752.608} C_VEL
LIN {X 0,Y 125.497,Z 374.611,A -85,B 0,C 180,E1 -25755.062,E2 -25755.062} C_VEL
LIN {X 0,Y 127.742,Z 384.857,A -85,B 0,C 180,E1 -25762.802,E2 -25762.802} C_VEL
LIN {X 0,Y 129.399,Z 387.929,A -85,B 0,C 180,E1 -25765.752,E2 -25765.752} C_VEL
LIN {X 0,Y 130.352,Z 389.407,A -85,B 0,C 180,E1 -25767.274,E2 -25767.274} C_VEL
LIN {X 0,Y 132.325,Z 392.9,A -85,B 0,C 180,E1 -25770.3,E2 -25770.3} C_VEL
LIN {X 0,Y 135.224,Z 399.337,A -85,B 0,C 180,E1 -25774.867,E2 -25774.867} C_VEL
LIN {X 0,Y 137.694,Z 405.416,A -85,B 0,C 180,E1 -25778.699,E2 -25778.699} C_VEL
LIN {X 0,Y 140.097,Z 413.516,A -85,B 0,C 180,E1 -25783.304,E2 -25783.304} C_VEL
LIN {X 0,Y 141.581,Z 421.266,A -85,B 0,C 180,E1 -25787.458,E2 -25787.458} C_VEL
LIN {X 0,Y 142.369,Z 428.863,A -85,B 0,C 180,E1 -25791.55,E2 -25791.55} C_VEL
LIN {X 0,Y 142.899,Z 437.595,A -85,B 0,C 180,E1 -25796.726,E2 -25796.726} C_VEL
LIN {X 0,Y 144.385,Z 443.831,A -85,B 0,C 180,E1 -25801.179,E2 -25801.179} C_VEL
LIN {X 0,Y 146.9,Z 448.767,A -85,B 0,C 180,E1 -25805.363,E2 -25805.363} C_VEL
LIN {X 0,Y 150.287,Z 452.725,A -85,B 0,C 180,E1 -25809.268,E2 -25809.268} C_VEL
LIN {X 0,Y 156.325,Z 456.965,A -85,B 0,C 180,E1 -25814.351,E2 -25814.351} C_VEL
LIN {X 0,Y 161,Z 459.128,A -85,B 0,C 180,E1 -25817.393,E2 -25817.393} C_VEL
LIN {X 0,Y 170.23,Z 461.658,A -85,B 0,C 180,E1 -25822.231,E2 -25822.231} C_VEL
LIN {X 0,Y 177.792,Z 462.797,A -85,B 0,C 180,E1 -25825.466,E2 -25825.466} C_VEL
LIN {X 0,Y 183.969,Z 463.196,A -85,B 0,C 180,E1 -25827.811,E2 -25827.811} C_VEL
LIN {X 0,Y 190.085,Z 463.187,A -85,B 0,C 180,E1 -25830,E2 -25830} C_VEL
LIN {X 0,Y 182.908,Z 463.133,A -85,B 0,C 180,E1 -25832.573,E2 -25832.573} C_VEL
LIN {X 0,Y 176.396,Z 462.652,A -85,B 0,C 180,E1 -25835.108,E2 -25835.108} C_VEL
LIN {X 0,Y 166.191,Z 460.74,A -85,B 0,C 180,E1 -25839.739,E2 -25839.739} C_VEL
LIN {X 0,Y 159.156,Z 458.371,A -85,B 0,C 180,E1 -25843.724,E2 -25843.724} C_VEL
LIN {X 0,Y 154.399,Z 455.931,A -85,B 0,C 180,E1 -25847.087,E2 -25847.087} C_VEL
LIN {X 0,Y 148.898,Z 451.364,A -85,B 0,C 180,E1 -25852.185,E2 -25852.185} C_VEL
LIN {X 0,Y 145.173,Z 445.636,A -85,B 0,C 180,E1 -25857.372,E2 -25857.372} C_VEL
LIN {X 0,Y 143.307,Z 439.753,A -85,B 0,C 180,E1 -25861.816,E2 -25861.816} C_VEL
LIN {X 0,Y 142.569,Z 434.233,A -85,B 0,C 180,E1 -25865.395,E2 -25865.395} C_VEL
LIN {X 0,Y 142.261,Z 427.426,A -85,B 0,C 180,E1 -25869.214,E2 -25869.214} C_VEL
LIN {X 0,Y 141.379,Z 420.148,A -85,B 0,C 180,E1 -25873.132,E2 -25873.132} C_VEL
LIN {X 0,Y 139.805,Z 412.503,A -85,B 0,C 180,E1 -25877.264,E2 -25877.264} C_VEL
LIN {X 0,Y 137.694,Z 405.414,A -85,B 0,C 180,E1 -25881.301,E2 -25881.301} C_VEL
LIN {X 0,Y 134.65,Z 398.003,A -85,B 0,C 180,E1 -25886.054,E2 -25886.054} C_VEL
LIN {X 0,Y 132.322,Z 392.908,A -85,B 0,C 180,E1 -25889.699,E2 -25889.699} C_VEL
LIN {X 0,Y 129.403,Z 387.919,A -85,B 0,C 180,E1 -25894.249,E2 -25894.249} C_VEL
LIN {X 0,Y 127.68,Z 384.68,A -85,B 0,C 180,E1 -25897.339,E2 -25897.339} C_VEL
LIN {X 0,Y 125.154,Z 381.415,A -85,B 0,C 180,E1 -25902.014,E2 -25902.014} C_VEL
LIN {X 0,Y 124.636,Z 379.92,A -85,B 0,C 180,E1 -25903.626,E2 -25903.626} C_VEL
LIN {X 0,Y 121.855,Z 376.77,A -85,B 0,C 180,E1 -25912.129,E2 -25912.129} C_VEL
LIN {X 0,Y 121.451,Z 374.269,A -85,B 0,C 180,E1 -25920.002,E2 -25920.002} C_VEL
LIN {X 0,Y 124.442,Z 379.42,A -85,B 0,C 180,E1 -25934.725,E2 -25934.725} C_VEL
LIN {X 0,Y 126.237,Z 383.8,A -85,B 0,C 180,E1 -25939.516,E2 -25939.516} C_VEL
LIN {X 0,Y 127.097,Z 385.015,A -85,B 0,C 180,E1 -25941.067,E2 -25941.067} C_VEL
LIN {X 0,Y 130.164,Z 391.107,A -85,B 0,C 180,E1 -25946.454,E2 -25946.454} C_VEL
LIN {X 0,Y 132.745,Z 397.911,A -85,B 0,C 180,E1 -25951.079,E2 -25951.079} C_VEL
LIN {X 0,Y 134.36,Z 402.486,A -85,B 0,C 180,E1 -25953.903,E2 -25953.903} C_VEL
LIN {X 0,Y 135.694,Z 407.902,A -85,B 0,C 180,E1 -25956.776,E2 -25956.776} C_VEL
LIN {X 0,Y 136.272,Z 413.308,A -85,B 0,C 180,E1 -25959.322,E2 -25959.322} C_VEL
LIN {X 0,Y 136.167,Z 421.089,A -85,B 0,C 180,E1 -25962.673,E2 -25962.673} C_VEL
LIN {X 0,Y 135.433,Z 427.76,A -85,B 0,C 180,E1 -25965.531,E2 -25965.531} C_VEL
LIN {X 0,Y 133.992,Z 435.365,A -85,B 0,C 180,E1 -25969.032,E2 -25969.032} C_VEL
LIN {X 0,Y 132.452,Z 440.293,A -85,B 0,C 180,E1 -25971.431,E2 -25971.431} C_VEL
LIN {X 0,Y 127.245,Z 448.623,A -85,B 0,C 180,E1 -25975.52,E2 -25975.52} C_VEL
LIN {X 0,Y 123.573,Z 454.286,A -85,B 0,C 180,E1 -25979.212,E2 -25979.212} C_VEL
LIN {X 0,Y 119.559,Z 459.777,A -85,B 0,C 180,E1 -25983.841,E2 -25983.841} C_VEL
LIN {X 0,Y 116.354,Z 464.103,A -85,B 0,C 180,E1 -25988.752,E2 -25988.752} C_VEL
LIN {X 0,Y 114.786,Z 466.476,A -85,B 0,C 180,E1 -25992.174,E2 -25992.174} C_VEL
LIN {X 0,Y 113.628,Z 468.282,A -85,B 0,C 180,E1 -25995.676,E2 -25995.676} C_VEL
LIN {X 0,Y 112.334,Z 470.744,A -85,B 0,C 180,E1 -26002.812,E2 -26002.812} C_VEL
LIN {X 0,Y 112.139,Z 471.34,A -85,B 0,C 180,E1 -26006.407,E2 -26006.407} C_VEL
LIN {X 0,Y 112.253,Z 471.501,A -85,B 0,C 180,E1 -26010,E2 -26010} C_VEL
LIN {X 0,Y 112.13,Z 471.339,A -85,B 0,C 180,E1 -26013.593,E2 -26013.593} C_VEL
LIN {X 0,Y 112.275,Z 470.742,A -85,B 0,C 180,E1 -26017.192,E2 -26017.192} C_VEL
LIN {X 0,Y 113.628,Z 468.282,A -85,B 0,C 180,E1 -26024.324,E2 -26024.324} C_VEL
LIN {X 0,Y 115.507,Z 465.322,A -85,B 0,C 180,E1 -26029.551,E2 -26029.551} C_VEL
LIN {X 0,Y 118.424,Z 461.331,A -85,B 0,C 180,E1 -26034.546,E2 -26034.546} C_VEL
LIN {X 0,Y 122.147,Z 456.201,A -85,B 0,C 180,E1 -26039.279,E2 -26039.279} C_VEL
LIN {X 0,Y 125.47,Z 451.256,A -85,B 0,C 180,E1 -26042.836,E2 -26042.836} C_VEL
LIN {X 0,Y 129.766,Z 444.617,A -85,B 0,C 180,E1 -26046.566,E2 -26046.566} C_VEL
LIN {X 0,Y 132.452,Z 440.293,A -85,B 0,C 180,E1 -26048.569,E2 -26048.569} C_VEL
LIN {X 0,Y 133.529,Z 437.011,A -85,B 0,C 180,E1 -26050.147,E2 -26050.147} C_VEL
LIN {X 0,Y 135.127,Z 429.708,A -85,B 0,C 180,E1 -26053.559,E2 -26053.559} C_VEL
LIN {X 0,Y 135.96,Z 423.35,A -85,B 0,C 180,E1 -26056.359,E2 -26056.359} C_VEL
LIN {X 0,Y 136.317,Z 416.342,A -85,B 0,C 180,E1 -26059.39,E2 -26059.39} C_VEL
LIN {X 0,Y 136.043,Z 410.157,A -85,B 0,C 180,E1 -26062.148,E2 -26062.148} C_VEL
LIN {X 0,Y 134.879,Z 404.392,A -85,B 0,C 180,E1 -26065.027,E2 -26065.027} C_VEL
LIN {X 0,Y 133.261,Z 399.036,A -85,B 0,C 180,E1 -26068.169,E2 -26068.169} C_VEL
LIN {X 0,Y 131.381,Z 394.423,A -85,B 0,C 180,E1 -26071.219,E2 -26071.219} C_VEL
LIN {X 0,Y 129.689,Z 390.277,A -85,B 0,C 180,E1 -26074.306,E2 -26074.306} C_VEL
LIN {X 0,Y 127.098,Z 385.014,A -85,B 0,C 180,E1 -26078.933,E2 -26078.933} C_VEL
LIN {X 0,Y 124.944,Z 380.924,A -85,B 0,C 180,E1 -26083.664,E2 -26083.664} C_VEL
LIN {X 0,Y 124.25,Z 379.298,A -85,B 0,C 180,E1 -26085.671,E2 -26085.671} C_VEL
LIN {X 0,Y 121.455,Z 374.253,A -85,B 0,C 180,E1 -26099.998,E2 -26099.998} C_VEL
LIN {X 0,Y 123.362,Z 378.54,A -85,B 0,C 180,E1 -26113.171,E2 -26113.171} C_VEL
LIN {X 0,Y 124.709,Z 380.212,A -85,B 0,C 180,E1 -26116.657,E2 -26116.657} C_VEL
LIN {X 0,Y 125.871,Z 382.601,A -85,B 0,C 180,E1 -26119.571,E2 -26119.571} C_VEL
LIN {X 0,Y 127.742,Z 384.857,A -85,B 0,C 180,E1 -26122.802,E2 -26122.802} C_VEL
LIN {X 0,Y 128.59,Z 388.049,A -85,B 0,C 180,E1 -26125.008,E2 -26125.008} C_VEL
LIN {X 0,Y 129.208,Z 394.394,A -85,B 0,C 180,E1 -26128.397,E2 -26128.397} C_VEL
LIN {X 0,Y 129.923,Z 402.047,A -85,B 0,C 180,E1 -26132.475,E2 -26132.475} C_VEL
LIN {X 0,Y 130.587,Z 404.235,A -85,B 0,C 180,E1 -26133.913,E2 -26133.913} C_VEL
LIN {X 0,Y 132.704,Z 410.35,A -85,B 0,C 180,E1 -26138.176,E2 -26138.176} C_VEL
LIN {X 0,Y 134.287,Z 416.683,A -85,B 0,C 180,E1 -26142.105,E2 -26142.105} C_VEL
LIN {X 0,Y 135.338,Z 422.555,A -85,B 0,C 180,E1 -26145.56,E2 -26145.56} C_VEL
LIN {X 0,Y 135.993,Z 429.703,A -85,B 0,C 180,E1 -26149.756,E2 -26149.756} C_VEL
LIN {X 0,Y 136.078,Z 437.318,A -85,B 0,C 180,E1 -26154.477,E2 -26154.477} C_VEL
LIN {X 0,Y 136.957,Z 443.637,A -85,B 0,C 180,E1 -26159.126,E2 -26159.126} C_VEL
LIN {X 0,Y 138.407,Z 447.962,A -85,B 0,C 180,E1 -26162.806,E2 -26162.806} C_VEL
LIN {X 0,Y 141.9,Z 452.996,A -85,B 0,C 180,E1 -26168.005,E2 -26168.005} C_VEL
LIN {X 0,Y 146.967,Z 456.972,A -85,B 0,C 180,E1 -26173.014,E2 -26173.014} C_VEL
LIN {X 0,Y 151.753,Z 459.39,A -85,B 0,C 180,E1 -26176.611,E2 -26176.611} C_VEL
LIN {X 0,Y 157.07,Z 461.097,A -85,B 0,C 180,E1 -26179.849,E2 -26179.849} C_VEL
LIN {X 0,Y 168.081,Z 463.062,A -85,B 0,C 180,E1 -26185.203,E2 -26185.203} C_VEL
LIN {X 0,Y 175.778,Z 463.528,A -85,B 0,C 180,E1 -26188.244,E2 -26188.244} C_VEL
LIN {X 0,Y 180.607,Z 463.444,A -85,B 0,C 180,E1 -26190,E2 -26190} C_VEL
LIN {X 0,Y 174.311,Z 463.461,A -85,B 0,C 180,E1 -26192.311,E2 -26192.311} C_VEL
LIN {X 0,Y 168.085,Z 463.061,A -85,B 0,C 180,E1 -26194.797,E2 -26194.797} C_VEL
LIN {X 0,Y 156.736,Z 461,A -85,B 0,C 180,E1 -26200.332,E2 -26200.332} C_VEL
LIN {X 0,Y 149.47,Z 458.341,A -85,B 0,C 180,E1 -26204.986,E2 -26204.986} C_VEL
LIN {X 0,Y 145.459,Z 456.067,A -85,B 0,C 180,E1 -26208.309,E2 -26208.309} C_VEL
LIN {X 0,Y 140.765,Z 451.607,A -85,B 0,C 180,E1 -26213.542,E2 -26213.542} C_VEL
LIN {X 0,Y 137.915,Z 446.632,A -85,B 0,C 180,E1 -26218.375,E2 -26218.375} C_VEL
LIN {X 0,Y 136.289,Z 440.02,A -85,B 0,C 180,E1 -26223.641,E2 -26223.641} C_VEL
LIN {X 0,Y 136.027,Z 434.455,A -85,B 0,C 180,E1 -26227.378,E2 -26227.378} C_VEL
LIN {X 0,Y 135.886,Z 428.014,A -85,B 0,C 180,E1 -26231.255,E2 -26231.255} C_VEL
LIN {X 0,Y 135.072,Z 421.027,A -85,B 0,C 180,E1 -26235.382,E2 -26235.382} C_VEL
LIN {X 0,Y 133.849,Z 414.7,A -85,B 0,C 180,E1 -26239.134,E2 -26239.134} C_VEL
LIN {X 0,Y 132.164,Z 408.727,A -85,B 0,C 180,E1 -26242.905,E2 -26242.905} C_VEL
LIN {X 0,Y 129.93,Z 402.617,A -85,B 0,C 180,E1 -26247.257,E2 -26247.257} C_VEL
LIN {X 0,Y 128.273,Z 398.527,A -85,B 0,C 180,E1 -26250.457,E2 -26250.457} C_VEL
LIN {X 0,Y 126.589,Z 395.087,A -85,B 0,C 180,E1 -26253.633,E2 -26253.633} C_VEL
LIN {X 0,Y 124.227,Z 390.563,A -85,B 0,C 180,E1 -26258.426,E2 -26258.426} C_VEL
LIN {X 0,Y 122.214,Z 387.276,A -85,B 0,C 180,E1 -26263.292,E2 -26263.292} C_VEL
LIN {X 0,Y 121.079,Z 385.413,A -85,B 0,C 180,E1 -26266.577,E2 -26266.577} C_VEL
LIN {X 0,Y 119.465,Z 381.229,A -85,B 0,C 180,E1 -26280.002,E2 -26280.002} C_VEL
LIN {X 0,Y 121.504,Z 385.69,A -85,B 0,C 180,E1 -26293.379,E2 -26293.379} C_VEL
LIN {X 0,Y 122.039,Z 386.773,A -85,B 0,C 180,E1 -26295.021,E2 -26295.021} C_VEL
LIN {X 0,Y 123.008,Z 389.446,A -85,B 0,C 180,E1 -26297.988,E2 -26297.988} C_VEL
LIN {X 0,Y 124.497,Z 392.425,A -85,B 0,C 180,E1 -26301.528,E2 -26301.528} C_VEL
LIN {X 0,Y 126.353,Z 396.792,A -85,B 0,C 180,E1 -26305.537,E2 -26305.537} C_VEL
LIN {X 0,Y 128.17,Z 402.243,A -85,B 0,C 180,E1 -26309.573,E2 -26309.573} C_VEL
LIN {X 0,Y 129.627,Z 407.171,A -85,B 0,C 180,E1 -26312.833,E2 -26312.833} C_VEL
LIN {X 0,Y 130.489,Z 411.566,A -85,B 0,C 180,E1 -26315.403,E2 -26315.403} C_VEL
LIN {X 0,Y 130.867,Z 418.038,A -85,B 0,C 180,E1 -26318.633,E2 -26318.633} C_VEL
LIN {X 0,Y 130.06,Z 426.538,A -85,B 0,C 180,E1 -26322.587,E2 -26322.587} C_VEL
LIN {X 0,Y 128.224,Z 435.368,A -85,B 0,C 180,E1 -26326.895,E2 -26326.895} C_VEL
LIN {X 0,Y 126.811,Z 440.091,A -85,B 0,C 180,E1 -26329.368,E2 -26329.368} C_VEL
LIN {X 0,Y 124.13,Z 444.421,A -85,B 0,C 180,E1 -26331.479,E2 -26331.479} C_VEL
LIN {X 0,Y 119.815,Z 450.65,A -85,B 0,C 180,E1 -26335.039,E2 -26335.039} C_VEL
LIN {X 0,Y 115.992,Z 456.005,A -85,B 0,C 180,E1 -26339.002,E2 -26339.002} C_VEL
LIN {X 0,Y 111.983,Z 461.135,A -85,B 0,C 180,E1 -26343.94,E2 -26343.94} C_VEL
LIN {X 0,Y 108.816,Z 465.126,A -85,B 0,C 180,E1 -26349.193,E2 -26349.193} C_VEL
LIN {X 0,Y 106.717,Z 468.085,A -85,B 0,C 180,E1 -26354.727,E2 -26354.727} C_VEL
LIN {X 0,Y 105.277,Z 470.547,A -85,B 0,C 180,E1 -26362.327,E2 -26362.327} C_VEL
LIN {X 0,Y 105.048,Z 471.144,A -85,B 0,C 180,E1 -26366.164,E2 -26366.164} C_VEL
LIN {X 0,Y 105.171,Z 471.306,A -85,B 0,C 180,E1 -26370,E2 -26370} C_VEL
LIN {X 0,Y 105.039,Z 471.143,A -85,B 0,C 180,E1 -26373.836,E2 -26373.836} C_VEL
LIN {X 0,Y 105.233,Z 470.546,A -85,B 0,C 180,E1 -26377.676,E2 -26377.676} C_VEL
LIN {X 0,Y 106.717,Z 468.085,A -85,B 0,C 180,E1 -26385.273,E2 -26385.273} C_VEL
LIN {X 0,Y 108.817,Z 465.126,A -85,B 0,C 180,E1 -26390.807,E2 -26390.807} C_VEL
LIN {X 0,Y 111.985,Z 461.135,A -85,B 0,C 180,E1 -26396.06,E2 -26396.06} C_VEL
LIN {X 0,Y 115.991,Z 456.005,A -85,B 0,C 180,E1 -26400.999,E2 -26400.999} C_VEL
LIN {X 0,Y 120.616,Z 449.583,A -85,B 0,C 180,E1 -26405.639,E2 -26405.639} C_VEL
LIN {X 0,Y 125.992,Z 441.661,A -85,B 0,C 180,E1 -26409.902,E2 -26409.902} C_VEL
LIN {X 0,Y 126.811,Z 440.091,A -85,B 0,C 180,E1 -26410.632,E2 -26410.632} C_VEL
LIN {X 0,Y 128.73,Z 433.286,A -85,B 0,C 180,E1 -26414.164,E2 -26414.164} C_VEL
LIN {X 0,Y 130.186,Z 425.431,A -85,B 0,C 180,E1 -26417.926,E2 -26417.926} C_VEL
LIN {X 0,Y 130.812,Z 417.093,A -85,B 0,C 180,E1 -26421.839,E2 -26421.839} C_VEL
LIN {X 0,Y 130.474,Z 411.596,A -85,B 0,C 180,E1 -26424.591,E2 -26424.591} C_VEL
LIN {X 0,Y 129.281,Z 405.814,A -85,B 0,C 180,E1 -26427.991,E2 -26427.991} C_VEL
LIN {X 0,Y 127.603,Z 400.354,A -85,B 0,C 180,E1 -26431.791,E2 -26431.791} C_VEL
LIN {X 0,Y 125.931,Z 395.925,A -85,B 0,C 180,E1 -26435.254,E2 -26435.254} C_VEL
LIN {X 0,Y 123.842,Z 390.889,A -85,B 0,C 180,E1 -26440.091,E2 -26440.091} C_VEL
LIN {X 0,Y 121.512,Z 385.664,A -85,B 0,C 180,E1 -26446.622,E2 -26446.622} C_VEL
LIN {X 0,Y 119.475,Z 381.198,A -85,B 0,C 180,E1 -26459.998,E2 -26459.998} C_VEL
LIN {X 0,Y 121.082,Z 385.404,A -85,B 0,C 180,E1 -26473.423,E2 -26473.423} C_VEL
LIN {X 0,Y 122.214,Z 387.276,A -85,B 0,C 180,E1 -26476.708,E2 -26476.708} C_VEL
LIN {X 0,Y 124.316,Z 390.829,A -85,B 0,C 180,E1 -26481.831,E2 -26481.831} C_VEL
LIN {X 0,Y 126.584,Z 395.101,A -85,B 0,C 180,E1 -26486.368,E2 -26486.368} C_VEL
LIN {X 0,Y 128.636,Z 399.578,A -85,B 0,C 180,E1 -26490.354,E2 -26490.354} C_VEL
LIN {X 0,Y 130.587,Z 404.235,A -85,B 0,C 180,E1 -26493.913,E2 -26493.913} C_VEL
LIN {X 0,Y 131.158,Z 406.483,A -85,B 0,C 180,E1 -26495.311,E2 -26495.311} C_VEL
LIN {X 0,Y 131.263,Z 409.065,A -85,B 0,C 180,E1 -26496.621,E2 -26496.621} C_VEL
LIN {X 0,Y 130.581,Z 414.686,A -85,B 0,C 180,E1 -26499.093,E2 -26499.093} C_VEL
LIN {X 0,Y 129.541,Z 420.37,A -85,B 0,C 180,E1 -26501.612,E2 -26501.612} C_VEL
LIN {X 0,Y 129.207,Z 424.174,A -85,B 0,C 180,E1 -26503.664,E2 -26503.664} C_VEL
LIN {X 0,Y 129.279,Z 425.31,A -85,B 0,C 180,E1 -26504.388,E2 -26504.388} C_VEL
LIN {X 0,Y 129.661,Z 431.72,A -85,B 0,C 180,E1 -26508.526,E2 -26508.526} C_VEL
LIN {X 0,Y 129.554,Z 437.542,A -85,B 0,C 180,E1 -26512.39,E2 -26512.39} C_VEL
LIN {X 0,Y 129.85,Z 443.868,A -85,B 0,C 180,E1 -26517.232,E2 -26517.232} C_VEL
LIN {X 0,Y 131.654,Z 450.028,A -85,B 0,C 180,E1 -26523.017,E2 -26523.017} C_VEL
LIN {X 0,Y 135.272,Z 454.885,A -85,B 0,C 180,E1 -26528.674,E2 -26528.674} C_VEL
LIN {X 0,Y 139.524,Z 458.015,A -85,B 0,C 180,E1 -26533.141,E2 -26533.141} C_VEL
LIN {X 0,Y 144.285,Z 460.232,A -85,B 0,C 180,E1 -26536.945,E2 -26536.945} C_VEL
LIN {X 0,Y 152.65,Z 462.455,A -85,B 0,C 180,E1 -26542.061,E2 -26542.061} C_VEL
LIN {X 0,Y 161.945,Z 463.562,A -85,B 0,C 180,E1 -26546.48,E2 -26546.48} C_VEL
LIN {X 0,Y 171.004,Z 463.704,A -85,B 0,C 180,E1 -26550,E2 -26550} C_VEL
LIN {X 0,Y 161.945,Z 463.561,A -85,B 0,C 180,E1 -26553.521,E2 -26553.521} C_VEL
LIN {X 0,Y 152.645,Z 462.455,A -85,B 0,C 180,E1 -26557.939,E2 -26557.939} C_VEL
LIN {X 0,Y 144.279,Z 460.239,A -85,B 0,C 180,E1 -26563.045,E2 -26563.045} C_VEL
LIN {X 0,Y 137.033,Z 456.415,A -85,B 0,C 180,E1 -26569.358,E2 -26569.358} C_VEL
LIN {X 0,Y 132.455,Z 451.348,A -85,B 0,C 180,E1 -26575.58,E2 -26575.58} C_VEL
LIN {X 0,Y 130.412,Z 446.54,A -85,B 0,C 180,E1 -26580.433,E2 -26580.433} C_VEL
LIN {X 0,Y 129.522,Z 440.435,A -85,B 0,C 180,E1 -26585.523,E2 -26585.523} C_VEL
LIN {X 0,Y 129.669,Z 434.385,A -85,B 0,C 180,E1 -26589.745,E2 -26589.745} C_VEL
LIN {X 0,Y 129.507,Z 428.21,A -85,B 0,C 180,E1 -26593.805,E2 -26593.805} C_VEL
LIN {X 0,Y 128.909,Z 422.107,A -85,B 0,C 180,E1 -26597.748,E2 -26597.748} C_VEL
LIN {X 0,Y 127.504,Z 414.759,A -85,B 0,C 180,E1 -26602.679,E2 -26602.679} C_VEL
LIN {X 0,Y 125.741,Z 409.036,A -85,B 0,C 180,E1 -26606.97,E2 -26606.97} C_VEL
LIN {X 0,Y 124.056,Z 404.056,A -85,B 0,C 180,E1 -26611.155,E2 -26611.155} C_VEL
LIN {X 0,Y 122.547,Z 400.6,A -85,B 0,C 180,E1 -26614.527,E2 -26614.527} C_VEL
LIN {X 0,Y 120.635,Z 396.36,A -85,B 0,C 180,E1 -26619.542,E2 -26619.542} C_VEL
LIN {X 0,Y 118.393,Z 392.229,A -85,B 0,C 180,E1 -26626.266,E2 -26626.266} C_VEL
LIN {X 0,Y 117.014,Z 389.964,A -85,B 0,C 180,E1 -26633.103,E2 -26633.103} C_VEL
LIN {X 0,Y 117.128,Z 388.046,A -85,B 0,C 180,E1 -26640.002,E2 -26640.002} C_VEL
LIN {X 0,Y 117.929,Z 391.25,A -85,B 0,C 180,E1 -26650.301,E2 -26650.301} C_VEL
LIN {X 0,Y 118.884,Z 392.628,A -85,B 0,C 180,E1 -26653.68,E2 -26653.68} C_VEL
LIN {X 0,Y 120.892,Z 398.08,A -85,B 0,C 180,E1 -26660.416,E2 -26660.416} C_VEL
LIN {X 0,Y 122.582,Z 403.443,A -85,B 0,C 180,E1 -26665.469,E2 -26665.469} C_VEL
LIN {X 0,Y 123.94,Z 408.133,A -85,B 0,C 180,E1 -26669.142,E2 -26669.142} C_VEL
LIN {X 0,Y 124.925,Z 412.775,A -85,B 0,C 180,E1 -26672.45,E2 -26672.45} C_VEL
LIN {X 0,Y 125.417,Z 417.523,A -85,B 0,C 180,E1 -26675.258,E2 -26675.258} C_VEL
LIN {X 0,Y 125.069,Z 422.998,A -85,B 0,C 180,E1 -26678.181,E2 -26678.181} C_VEL
LIN {X 0,Y 124.024,Z 429.474,A -85,B 0,C 180,E1 -26681.47,E2 -26681.47} C_VEL
LIN {X 0,Y 122.101,Z 436.99,A -85,B 0,C 180,E1 -26685.445,E2 -26685.445} C_VEL
LIN {X 0,Y 120.554,Z 441.462,A -85,B 0,C 180,E1 -26687.901,E2 -26687.901} C_VEL
LIN {X 0,Y 114.846,Z 449.385,A -85,B 0,C 180,E1 -26692.27,E2 -26692.27} C_VEL
LIN {X 0,Y 109.948,Z 455.808,A -85,B 0,C 180,E1 -26697.089,E2 -26697.089} C_VEL
LIN {X 0,Y 105.631,Z 460.939,A -85,B 0,C 180,E1 -26702.242,E2 -26702.242} C_VEL
LIN {X 0,Y 102.193,Z 464.929,A -85,B 0,C 180,E1 -26707.775,E2 -26707.775} C_VEL
LIN {X 0,Y 99.841,Z 467.888,A -85,B 0,C 180,E1 -26713.646,E2 -26713.646} C_VEL
LIN {X 0,Y 98.224,Z 470.351,A -85,B 0,C 180,E1 -26721.773,E2 -26721.773} C_VEL
LIN {X 0,Y 97.954,Z 470.947,A -85,B 0,C 180,E1 -26725.886,E2 -26725.886} C_VEL
LIN {X 0,Y 98.077,Z 471.11,A -85,B 0,C 180,E1 -26730,E2 -26730} C_VEL
LIN {X 0,Y 97.945,Z 470.947,A -85,B 0,C 180,E1 -26734.115,E2 -26734.115} C_VEL
LIN {X 0,Y 98.19,Z 470.35,A -85,B 0,C 180,E1 -26738.23,E2 -26738.23} C_VEL
LIN {X 0,Y 99.841,Z 467.888,A -85,B 0,C 180,E1 -26746.354,E2 -26746.354} C_VEL
LIN {X 0,Y 102.194,Z 464.929,A -85,B 0,C 180,E1 -26752.225,E2 -26752.225} C_VEL
LIN {X 0,Y 105.632,Z 460.939,A -85,B 0,C 180,E1 -26757.757,E2 -26757.757} C_VEL
LIN {X 0,Y 109.95,Z 455.808,A -85,B 0,C 180,E1 -26762.91,E2 -26762.91} C_VEL
LIN {X 0,Y 114.884,Z 449.386,A -85,B 0,C 180,E1 -26767.716,E2 -26767.716} C_VEL
LIN {X 0,Y 120.551,Z 441.462,A -85,B 0,C 180,E1 -26772.101,E2 -26772.101} C_VEL
LIN {X 0,Y 122.89,Z 434.39,A -85,B 0,C 180,E1 -26776.018,E2 -26776.018} C_VEL
LIN {X 0,Y 124.779,Z 425.704,A -85,B 0,C 180,E1 -26780.477,E2 -26780.477} C_VEL
LIN {X 0,Y 125.438,Z 418.557,A -85,B 0,C 180,E1 -26784.152,E2 -26784.152} C_VEL
LIN {X 0,Y 124.925,Z 412.775,A -85,B 0,C 180,E1 -26787.55,E2 -26787.55} C_VEL
LIN {X 0,Y 123.963,Z 408.044,A -85,B 0,C 180,E1 -26790.885,E2 -26790.885} C_VEL
LIN {X 0,Y 122.029,Z 401.489,A -85,B 0,C 180,E1 -26796.223,E2 -26796.223} C_VEL
LIN {X 0,Y 120.912,Z 398.032,A -85,B 0,C 180,E1 -26799.587,E2 -26799.587} C_VEL
LIN {X 0,Y 118.884,Z 392.626,A -85,B 0,C 180,E1 -26806.32,E2 -26806.32} C_VEL
LIN {X 0,Y 117.248,Z 390.2,A -85,B 0,C 180,E1 -26813.113,E2 -26813.113} C_VEL
LIN {X 0,Y 117.145,Z 388.002,A -85,B 0,C 180,E1 -26819.998,E2 -26819.998} C_VEL
LIN {X 0,Y 117.547,Z 390.973,A -85,B 0,C 180,E1 -26830.331,E2 -26830.331} C_VEL
LIN {X 0,Y 118.392,Z 392.23,A -85,B 0,C 180,E1 -26833.734,E2 -26833.734} C_VEL
LIN {X 0,Y 120.623,Z 396.388,A -85,B 0,C 180,E1 -26840.46,E2 -26840.46} C_VEL
LIN {X 0,Y 122.533,Z 400.63,A -85,B 0,C 180,E1 -26845.476,E2 -26845.476} C_VEL
LIN {X 0,Y 124.059,Z 404.05,A -85,B 0,C 180,E1 -26848.845,E2 -26848.845} C_VEL
LIN {X 0,Y 126.474,Z 411.185,A -85,B 0,C 180,E1 -26854.719,E2 -26854.719} C_VEL
LIN {X 0,Y 127.86,Z 416.53,A -85,B 0,C 180,E1 -26858.568,E2 -26858.568} C_VEL
LIN {X 0,Y 128.917,Z 422.101,A -85,B 0,C 180,E1 -26862.253,E2 -26862.253} C_VEL
LIN {X 0,Y 129.279,Z 425.31,A -85,B 0,C 180,E1 -26864.388,E2 -26864.388} C_VEL
LIN {X 0,Y 128.987,Z 429.01,A -85,B 0,C 180,E1 -26866.442,E2 -26866.442} C_VEL
LIN {X 0,Y 127.582,Z 432.915,A -85,B 0,C 180,E1 -26868.391,E2 -26868.391} C_VEL
LIN {X 0,Y 123.597,Z 441.469,A -85,B 0,C 180,E1 -26873.114,E2 -26873.114} C_VEL
LIN {X 0,Y 123.006,Z 444.456,A -85,B 0,C 180,E1 -26875.477,E2 -26875.477} C_VEL
LIN {X 0,Y 123.613,Z 448.428,A -85,B 0,C 180,E1 -26879.224,E2 -26879.224} C_VEL
LIN {X 0,Y 125.213,Z 452.652,A -85,B 0,C 180,E1 -26883.899,E2 -26883.899} C_VEL
LIN {X 0,Y 128.163,Z 456.295,A -85,B 0,C 180,E1 -26888.778,E2 -26888.778} C_VEL
LIN {X 0,Y 133.719,Z 459.903,A -85,B 0,C 180,E1 -26894.764,E2 -26894.764} C_VEL
LIN {X 0,Y 142.306,Z 462.549,A -85,B 0,C 180,E1 -26901.006,E2 -26901.006} C_VEL
LIN {X 0,Y 148.797,Z 463.587,A -85,B 0,C 180,E1 -26904.58,E2 -26904.58} C_VEL
LIN {X 0,Y 154.86,Z 463.992,A -85,B 0,C 180,E1 -26907.399,E2 -26907.399} C_VEL
LIN {X 0,Y 161.319,Z 463.966,A -85,B 0,C 180,E1 -26910,E2 -26910} C_VEL
LIN {X 0,Y 154.775,Z 463.987,A -85,B 0,C 180,E1 -26912.635,E2 -26912.635} C_VEL
LIN {X 0,Y 148.307,Z 463.553,A -85,B 0,C 180,E1 -26915.661,E2 -26915.661} C_VEL
LIN {X 0,Y 138.081,Z 461.516,A -85,B 0,C 180,E1 -26921.747,E2 -26921.747} C_VEL
LIN {X 0,Y 132.098,Z 459.039,A -85,B 0,C 180,E1 -26926.74,E2 -26926.74} C_VEL
LIN {X 0,Y 127.134,Z 455.127,A -85,B 0,C 180,E1 -26932.766,E2 -26932.766} C_VEL
LIN {X 0,Y 124.965,Z 452.089,A -85,B 0,C 180,E1 -26936.738,E2 -26936.738} C_VEL
LIN {X 0,Y 123.201,Z 446.325,A -85,B 0,C 180,E1 -26942.813,E2 -26942.813} C_VEL
LIN {X 0,Y 123.007,Z 440.445,A -85,B 0,C 180,E1 -26947.886,E2 -26947.886} C_VEL
LIN {X 0,Y 123.402,Z 434.571,A -85,B 0,C 180,E1 -26952.239,E2 -26952.239} C_VEL
LIN {X 0,Y 123.254,Z 428.198,A -85,B 0,C 180,E1 -26956.826,E2 -26956.826} C_VEL
LIN {X 0,Y 122.707,Z 422.502,A -85,B 0,C 180,E1 -26960.951,E2 -26960.951} C_VEL
LIN {X 0,Y 121.535,Z 416.329,A -85,B 0,C 180,E1 -26965.672,E2 -26965.672} C_VEL
LIN {X 0,Y 120.061,Z 411.229,A -85,B 0,C 180,E1 -26970.165,E2 -26970.165} C_VEL
LIN {X 0,Y 119.529,Z 409.279,A -85,B 0,C 180,E1 -26971.943,E2 -26971.943} C_VEL
LIN {X 0,Y 118.398,Z 406.061,A -85,B 0,C 180,E1 -26975.45,E2 -26975.45} C_VEL
LIN {X 0,Y 116.691,Z 401.97,A -85,B 0,C 180,E1 -26980.657,E2 -26980.657} C_VEL
LIN {X 0,Y 115.384,Z 398.917,A -85,B 0,C 180,E1 -26985.901,E2 -26985.901} C_VEL
LIN {X 0,Y 114.162,Z 396.54,A -85,B 0,C 180,E1 -26992.93,E2 -26992.93} C_VEL
LIN {X 0,Y 114.283,Z 394.664,A -85,B 0,C 180,E1 -27000.002,E2 -27000.002} C_VEL
LIN {X 0,Y 115.075,Z 397.888,A -85,B 0,C 180,E1 -27010.559,E2 -27010.559} C_VEL
LIN {X 0,Y 115.789,Z 399.698,A -85,B 0,C 180,E1 -27014.053,E2 -27014.053} C_VEL
LIN {X 0,Y 116.969,Z 403.56,A -85,B 0,C 180,E1 -27019.299,E2 -27019.299} C_VEL
LIN {X 0,Y 118.381,Z 408.811,A -85,B 0,C 180,E1 -27024.557,E2 -27024.557} C_VEL
LIN {X 0,Y 119.645,Z 415.271,A -85,B 0,C 180,E1 -27029.955,E2 -27029.955} C_VEL
LIN {X 0,Y 120.033,Z 420.063,A -85,B 0,C 180,E1 -27033.282,E2 -27033.282} C_VEL
LIN {X 0,Y 119.594,Z 425.36,A -85,B 0,C 180,E1 -27036.338,E2 -27036.338} C_VEL
LIN {X 0,Y 117.982,Z 432.54,A -85,B 0,C 180,E1 -27040.309,E2 -27040.309} C_VEL
LIN {X 0,Y 115.678,Z 439.671,A -85,B 0,C 180,E1 -27044.45,E2 -27044.45} C_VEL
LIN {X 0,Y 114.332,Z 442.65,A -85,B 0,C 180,E1 -27046.248,E2 -27046.248} C_VEL
LIN {X 0,Y 109.293,Z 449.188,A -85,B 0,C 180,E1 -27049.981,E2 -27049.981} C_VEL
LIN {X 0,Y 105.69,Z 453.693,A -85,B 0,C 180,E1 -27053.24,E2 -27053.24} C_VEL
LIN {X 0,Y 100.77,Z 459.186,A -85,B 0,C 180,E1 -27058.462,E2 -27058.462} C_VEL
LIN {X 0,Y 96.776,Z 463.515,A -85,B 0,C 180,E1 -27064.169,E2 -27064.169} C_VEL
LIN {X 0,Y 94.607,Z 465.884,A -85,B 0,C 180,E1 -27068.196,E2 -27068.196} C_VEL
LIN {X 0,Y 93.015,Z 467.691,A -85,B 0,C 180,E1 -27072.408,E2 -27072.408} C_VEL
LIN {X 0,Y 91.176,Z 470.154,A -85,B 0,C 180,E1 -27081.132,E2 -27081.132} C_VEL
LIN {X 0,Y 90.883,Z 470.752,A -85,B 0,C 180,E1 -27085.565,E2 -27085.565} C_VEL
LIN {X 0,Y 90.976,Z 470.914,A -85,B 0,C 180,E1 -27090,E2 -27090} C_VEL
LIN {X 0,Y 90.875,Z 470.752,A -85,B 0,C 180,E1 -27094.436,E2 -27094.436} C_VEL
LIN {X 0,Y 91.15,Z 470.154,A -85,B 0,C 180,E1 -27098.871,E2 -27098.871} C_VEL
LIN {X 0,Y 93.015,Z 467.691,A -85,B 0,C 180,E1 -27107.592,E2 -27107.592} C_VEL
LIN {X 0,Y 95.622,Z 464.732,A -85,B 0,C 180,E1 -27113.843,E2 -27113.843} C_VEL
LIN {X 0,Y 99.368,Z 460.742,A -85,B 0,C 180,E1 -27119.675,E2 -27119.675} C_VEL
LIN {X 0,Y 104.026,Z 455.611,A -85,B 0,C 180,E1 -27125.048,E2 -27125.048} C_VEL
LIN {X 0,Y 108.452,Z 450.245,A -85,B 0,C 180,E1 -27129.288,E2 -27129.288} C_VEL
LIN {X 0,Y 113.3,Z 444.027,A -85,B 0,C 180,E1 -27133.026,E2 -27133.026} C_VEL
LIN {X 0,Y 114.336,Z 442.651,A -85,B 0,C 180,E1 -27133.75,E2 -27133.75} C_VEL
LIN {X 0,Y 116.685,Z 436.699,A -85,B 0,C 180,E1 -27137.293,E2 -27137.293} C_VEL
LIN {X 0,Y 118.358,Z 430.992,A -85,B 0,C 180,E1 -27140.527,E2 -27140.527} C_VEL
LIN {X 0,Y 119.629,Z 424.744,A -85,B 0,C 180,E1 -27144.019,E2 -27144.019} C_VEL
LIN {X 0,Y 120.041,Z 420.063,A -85,B 0,C 180,E1 -27146.712,E2 -27146.712} C_VEL
LIN {X 0,Y 119.836,Z 416.564,A -85,B 0,C 180,E1 -27149.123,E2 -27149.123} C_VEL
LIN {X 0,Y 118.808,Z 410.765,A -85,B 0,C 180,E1 -27153.659,E2 -27153.659} C_VEL
LIN {X 0,Y 117.915,Z 406.921,A -85,B 0,C 180,E1 -27157.184,E2 -27157.184} C_VEL
LIN {X 0,Y 116.997,Z 403.507,A -85,B 0,C 180,E1 -27160.706,E2 -27160.706} C_VEL
LIN {X 0,Y 115.762,Z 399.449,A -85,B 0,C 180,E1 -27166.256,E2 -27166.256} C_VEL
LIN {X 0,Y 115.072,Z 397.893,A -85,B 0,C 180,E1 -27169.44,E2 -27169.44} C_VEL
LIN {X 0,Y 114.307,Z 394.609,A -85,B 0,C 180,E1 -27179.998,E2 -27179.998} C_VEL
LIN {X 0,Y 114.918,Z 398.037,A -85,B 0,C 180,E1 -27191.903,E2 -27191.903} C_VEL
LIN {X 0,Y 115.729,Z 399.901,A -85,B 0,C 180,E1 -27195.857,E2 -27195.857} C_VEL
LIN {X 0,Y 117.204,Z 403.258,A -85,B 0,C 180,E1 -27201.085,E2 -27201.085} C_VEL
LIN {X 0,Y 118.394,Z 406.068,A -85,B 0,C 180,E1 -27204.55,E2 -27204.55} C_VEL
LIN {X 0,Y 119.557,Z 409.371,A -85,B 0,C 180,E1 -27208.146,E2 -27208.146} C_VEL
LIN {X 0,Y 121.202,Z 415.037,A -85,B 0,C 180,E1 -27213.201,E2 -27213.201} C_VEL
LIN {X 0,Y 122.516,Z 421.175,A -85,B 0,C 180,E1 -27218.069,E2 -27218.069} C_VEL
LIN {X 0,Y 123.28,Z 428.159,A -85,B 0,C 180,E1 -27223.162,E2 -27223.162} C_VEL
LIN {X 0,Y 123.383,Z 434.596,A -85,B 0,C 180,E1 -27227.77,E2 -27227.77} C_VEL
LIN {X 0,Y 122.999,Z 441.753,A -85,B 0,C 180,E1 -27233.122,E2 -27233.122} C_VEL
LIN {X 0,Y 123.006,Z 444.456,A -85,B 0,C 180,E1 -27235.477,E2 -27235.477} C_VEL
LIN {X 0,Y 122.509,Z 446.507,A -85,B 0,C 180,E1 -27237.095,E2 -27237.095} C_VEL
LIN {X 0,Y 118.321,Z 452.97,A -85,B 0,C 180,E1 -27242.377,E2 -27242.377} C_VEL
LIN {X 0,Y 118.376,Z 454.362,A -85,B 0,C 180,E1 -27244.153,E2 -27244.153} C_VEL
LIN {X 0,Y 121.589,Z 457.966,A -85,B 0,C 180,E1 -27249.708,E2 -27249.708} C_VEL
LIN {X 0,Y 124.95,Z 460.154,A -85,B 0,C 180,E1 -27253.666,E2 -27253.666} C_VEL
LIN {X 0,Y 129.443,Z 461.925,A -85,B 0,C 180,E1 -27257.758,E2 -27257.758} C_VEL
LIN {X 0,Y 139.23,Z 463.849,A -85,B 0,C 180,E1 -27264.206,E2 -27264.206} C_VEL
LIN {X 0,Y 147.645,Z 464.336,A -85,B 0,C 180,E1 -27268.345,E2 -27268.345} C_VEL
LIN {X 0,Y 151.581,Z 464.229,A -85,B 0,C 180,E1 -27270,E2 -27270} C_VEL
LIN {X 0,Y 141.052,Z 463.978,A -85,B 0,C 180,E1 -27274.809,E2 -27274.809} C_VEL
LIN {X 0,Y 133.773,Z 462.977,A -85,B 0,C 180,E1 -27279.068,E2 -27279.068} C_VEL
LIN {X 0,Y 129.008,Z 461.772,A -85,B 0,C 180,E1 -27282.586,E2 -27282.586} C_VEL
LIN {X 0,Y 123.21,Z 459.094,A -85,B 0,C 180,E1 -27288.282,E2 -27288.282} C_VEL
LIN {X 0,Y 119.083,Z 455.369,A -85,B 0,C 180,E1 -27294.401,E2 -27294.401} C_VEL
LIN {X 0,Y 116.878,Z 450.688,A -85,B 0,C 180,E1 -27300.525,E2 -27300.525} C_VEL
LIN {X 0,Y 116.266,Z 445.438,A -85,B 0,C 180,E1 -27306.112,E2 -27306.112} C_VEL
LIN {X 0,Y 116.879,Z 439.324,A -85,B 0,C 180,E1 -27311.409,E2 -27311.409} C_VEL
LIN {X 0,Y 117.183,Z 434.896,A -85,B 0,C 180,E1 -27314.996,E2 -27314.996} C_VEL
LIN {X 0,Y 117.17,Z 428.499,A -85,B 0,C 180,E1 -27320.064,E2 -27320.064} C_VEL
LIN {X 0,Y 116.588,Z 422.472,A -85,B 0,C 180,E1 -27325.066,E2 -27325.066} C_VEL
LIN {X 0,Y 115.725,Z 418.183,A -85,B 0,C 180,E1 -27328.922,E2 -27328.922} C_VEL
LIN {X 0,Y 114.773,Z 414.037,A -85,B 0,C 180,E1 -27333.21,E2 -27333.21} C_VEL
LIN {X 0,Y 113.391,Z 409.774,A -85,B 0,C 180,E1 -27338.388,E2 -27338.388} C_VEL
LIN {X 0,Y 112.268,Z 406.501,A -85,B 0,C 180,E1 -27343.64,E2 -27343.64} C_VEL
LIN {X 0,Y 111.964,Z 405.459,A -85,B 0,C 180,E1 -27345.461,E2 -27345.461} C_VEL
LIN {X 0,Y 111.305,Z 403.964,A -85,B 0,C 180,E1 -27349.083,E2 -27349.083} C_VEL
LIN {X 0,Y 111.13,Z 401.134,A -85,B 0,C 180,E1 -27360.002,E2 -27360.002} C_VEL
LIN {X 0,Y 111.702,Z 404.379,A -85,B 0,C 180,E1 -27370.882,E2 -27370.882} C_VEL
LIN {X 0,Y 111.996,Z 405.149,A -85,B 0,C 180,E1 -27372.536,E2 -27372.536} C_VEL
LIN {X 0,Y 112.951,Z 408.94,A -85,B 0,C 180,E1 -27378.128,E2 -27378.128} C_VEL
LIN {X 0,Y 113.841,Z 413.948,A -85,B 0,C 180,E1 -27383.66,E2 -27383.66} C_VEL
LIN {X 0,Y 114.48,Z 418.445,A -85,B 0,C 180,E1 -27387.731,E2 -27387.731} C_VEL
LIN {X 0,Y 114.72,Z 422.389,A -85,B 0,C 180,E1 -27390.944,E2 -27390.944} C_VEL
LIN {X 0,Y 114.384,Z 426.371,A -85,B 0,C 180,E1 -27393.574,E2 -27393.574} C_VEL
LIN {X 0,Y 112.497,Z 433.796,A -85,B 0,C 180,E1 -27398.052,E2 -27398.052} C_VEL
LIN {X 0,Y 109.757,Z 441.043,A -85,B 0,C 180,E1 -27402.577,E2 -27402.577} C_VEL
LIN {X 0,Y 108.208,Z 443.831,A -85,B 0,C 180,E1 -27404.403,E2 -27404.403} C_VEL
LIN {X 0,Y 102.821,Z 450.263,A -85,B 0,C 180,E1 -27408.339,E2 -27408.339} C_VEL
LIN {X 0,Y 98.265,Z 455.414,A -85,B 0,C 180,E1 -27412.56,E2 -27412.56} C_VEL
LIN {X 0,Y 93.218,Z 460.544,A -85,B 0,C 180,E1 -27418.146,E2 -27418.146} C_VEL
LIN {X 0,Y 89.146,Z 464.536,A -85,B 0,C 180,E1 -27424.304,E2 -27424.304} C_VEL
LIN {X 0,Y 86.247,Z 467.494,A -85,B 0,C 180,E1 -27430.977,E2 -27430.977} C_VEL
LIN {X 0,Y 84.156,Z 469.958,A -85,B 0,C 180,E1 -27440.385,E2 -27440.385} C_VEL
LIN {X 0,Y 83.798,Z 470.556,A -85,B 0,C 180,E1 -27445.189,E2 -27445.189} C_VEL
LIN {X 0,Y 83.883,Z 470.719,A -85,B 0,C 180,E1 -27450,E2 -27450} C_VEL
LIN {X 0,Y 83.791,Z 470.556,A -85,B 0,C 180,E1 -27454.811,E2 -27454.811} C_VEL
LIN {X 0,Y 84.137,Z 469.958,A -85,B 0,C 180,E1 -27459.617,E2 -27459.617} C_VEL
LIN {X 0,Y 86.247,Z 467.494,A -85,B 0,C 180,E1 -27469.023,E2 -27469.023} C_VEL
LIN {X 0,Y 89.146,Z 464.536,A -85,B 0,C 180,E1 -27475.696,E2 -27475.696} C_VEL
LIN {X 0,Y 93.219,Z 460.544,A -85,B 0,C 180,E1 -27481.853,E2 -27481.853} C_VEL
LIN {X 0,Y 98.263,Z 455.414,A -85,B 0,C 180,E1 -27487.441,E2 -27487.441} C_VEL
LIN {X 0,Y 102.839,Z 450.263,A -85,B 0,C 180,E1 -27491.652,E2 -27491.652} C_VEL
LIN {X 0,Y 108.197,Z 443.83,A -85,B 0,C 180,E1 -27495.603,E2 -27495.603} C_VEL
LIN {X 0,Y 109.724,Z 441.042,A -85,B 0,C 180,E1 -27497.442,E2 -27497.442} C_VEL
LIN {X 0,Y 112.482,Z 433.796,A -85,B 0,C 180,E1 -27501.957,E2 -27501.957} C_VEL
LIN {X 0,Y 114.097,Z 427.547,A -85,B 0,C 180,E1 -27505.696,E2 -27505.696} C_VEL
LIN {X 0,Y 114.675,Z 424.204,A -85,B 0,C 180,E1 -27507.791,E2 -27507.791} C_VEL
LIN {X 0,Y 114.635,Z 420.373,A -85,B 0,C 180,E1 -27510.627,E2 -27510.627} C_VEL
LIN {X 0,Y 114.188,Z 415.927,A -85,B 0,C 180,E1 -27514.478,E2 -27514.478} C_VEL
LIN {X 0,Y 113.512,Z 412.087,A -85,B 0,C 180,E1 -27518.234,E2 -27518.234} C_VEL
LIN {X 0,Y 112.977,Z 408.899,A -85,B 0,C 180,E1 -27521.876,E2 -27521.876} C_VEL
LIN {X 0,Y 111.999,Z 405.14,A -85,B 0,C 180,E1 -27527.47,E2 -27527.47} C_VEL
LIN {X 0,Y 111.144,Z 403.153,A -85,B 0,C 180,E1 -27532.733,E2 -27532.733} C_VEL
LIN {X 0,Y 111.169,Z 401.063,A -85,B 0,C 180,E1 -27539.998,E2 -27539.998} C_VEL
LIN {X 0,Y 111.304,Z 403.965,A -85,B 0,C 180,E1 -27550.917,E2 -27550.917} C_VEL
LIN {X 0,Y 111.959,Z 405.471,A -85,B 0,C 180,E1 -27554.54,E2 -27554.54} C_VEL
LIN {X 0,Y 113.081,Z 408.74,A -85,B 0,C 180,E1 -27560.176,E2 -27560.176} C_VEL
LIN {X 0,Y 113.922,Z 411.286,A -85,B 0,C 180,E1 -27563.638,E2 -27563.638} C_VEL
LIN {X 0,Y 115.085,Z 415.279,A -85,B 0,C 180,E1 -27568.135,E2 -27568.135} C_VEL
LIN {X 0,Y 116.163,Z 420.25,A -85,B 0,C 180,E1 -27572.989,E2 -27572.989} C_VEL
LIN {X 0,Y 116.849,Z 424.81,A -85,B 0,C 180,E1 -27576.972,E2 -27576.972} C_VEL
LIN {X 0,Y 117.253,Z 430.154,A -85,B 0,C 180,E1 -27581.246,E2 -27581.246} C_VEL
LIN {X 0,Y 117.159,Z 436.244,A -85,B 0,C 180,E1 -27586.039,E2 -27586.039} C_VEL
LIN {X 0,Y 116.463,Z 443.084,A -85,B 0,C 180,E1 -27591.67,E2 -27591.67} C_VEL
LIN {X 0,Y 116.555,Z 449.057,A -85,B 0,C 180,E1 -27597.579,E2 -27597.579} C_VEL
LIN {X 0,Y 118.008,Z 453.763,A -85,B 0,C 180,E1 -27603.29,E2 -27603.29} C_VEL
LIN {X 0,Y 118.376,Z 454.362,A -85,B 0,C 180,E1 -27604.153,E2 -27604.153} C_VEL
LIN {X 0,Y 119.064,Z 456.381,A -85,B 0,C 180,E1 -27606.839,E2 -27606.839} C_VEL
LIN {X 0,Y 119.167,Z 459.416,A -85,B 0,C 180,E1 -27611.385,E2 -27611.385} C_VEL
LIN {X 0,Y 120.219,Z 461.845,A -85,B 0,C 180,E1 -27615.924,E2 -27615.924} C_VEL
LIN {X 0,Y 122.316,Z 462.753,A -85,B 0,C 180,E1 -27618.472,E2 -27618.472} C_VEL
LIN {X 0,Y 129.764,Z 464.111,A -85,B 0,C 180,E1 -27623.782,E2 -27623.782} C_VEL
LIN {X 0,Y 140.563,Z 464.528,A -85,B 0,C 180,E1 -27629.429,E2 -27629.429} C_VEL
LIN {X 0,Y 141.882,Z 464.492,A -85,B 0,C 180,E1 -27630,E2 -27630} C_VEL
LIN {X 0,Y 133.832,Z 464.404,A -85,B 0,C 180,E1 -27633.864,E2 -27633.864} C_VEL
LIN {X 0,Y 127.613,Z 463.844,A -85,B 0,C 180,E1 -27637.572,E2 -27637.572} C_VEL
LIN {X 0,Y 120.081,Z 462.025,A -85,B 0,C 180,E1 -27643.539,E2 -27643.539} C_VEL
LIN {X 0,Y 114.787,Z 459.368,A -85,B 0,C 180,E1 -27649.633,E2 -27649.633} C_VEL
LIN {X 0,Y 112.229,Z 457.053,A -85,B 0,C 180,E1 -27654.019,E2 -27654.019} C_VEL
LIN {X 0,Y 110.037,Z 452.558,A -85,B 0,C 180,E1 -27660.727,E2 -27660.727} C_VEL
LIN {X 0,Y 109.67,Z 446.779,A -85,B 0,C 180,E1 -27667.502,E2 -27667.502} C_VEL
LIN {X 0,Y 110.597,Z 440.886,A -85,B 0,C 180,E1 -27673.087,E2 -27673.087} C_VEL
LIN {X 0,Y 111.147,Z 434.923,A -85,B 0,C 180,E1 -27678.385,E2 -27678.385} C_VEL
LIN {X 0,Y 111.234,Z 429.658,A -85,B 0,C 180,E1 -27683.116,E2 -27683.116} C_VEL
LIN {X 0,Y 110.824,Z 424.615,A -85,B 0,C 180,E1 -27687.839,E2 -27687.839} C_VEL
LIN {X 0,Y 109.986,Z 419.406,A -85,B 0,C 180,E1 -27693.455,E2 -27693.455} C_VEL
LIN {X 0,Y 109.11,Z 415.489,A -85,B 0,C 180,E1 -27698.671,E2 -27698.671} C_VEL
LIN {X 0,Y 108.353,Z 412.791,A -85,B 0,C 180,E1 -27703.032,E2 -27703.032} C_VEL
LIN {X 0,Y 107.585,Z 410.221,A -85,B 0,C 180,E1 -27708.7,E2 -27708.7} C_VEL
LIN {X 0,Y 107.268,Z 408.249,A -85,B 0,C 180,E1 -27716.245,E2 -27716.245} C_VEL
LIN {X 0,Y 107.688,Z 407.43,A -85,B 0,C 180,E1 -27720.002,E2 -27720.002} C_VEL
LIN {X 0,Y 107.579,Z 409.415,A -85,B 0,C 180,E1 -27727.51,E2 -27727.51} C_VEL
LIN {X 0,Y 108.038,Z 410.678,A -85,B 0,C 180,E1 -27731.256,E2 -27731.256} C_VEL
LIN {X 0,Y 108.619,Z 414.113,A -85,B 0,C 180,E1 -27736.93,E2 -27736.93} C_VEL
LIN {X 0,Y 109.164,Z 418.967,A -85,B 0,C 180,E1 -27742.725,E2 -27742.725} C_VEL
LIN {X 0,Y 109.448,Z 424.138,A -85,B 0,C 180,E1 -27747.748,E2 -27747.748} C_VEL
LIN {X 0,Y 109.131,Z 428.107,A -85,B 0,C 180,E1 -27751.013,E2 -27751.013} C_VEL
LIN {X 0,Y 107.974,Z 432.456,A -85,B 0,C 180,E1 -27753.883,E2 -27753.883} C_VEL
LIN {X 0,Y 105.333,Z 439.24,A -85,B 0,C 180,E1 -27758.374,E2 -27758.374} C_VEL
LIN {X 0,Y 103.205,Z 443.628,A -85,B 0,C 180,E1 -27761.49,E2 -27761.49} C_VEL
LIN {X 0,Y 98.797,Z 448.795,A -85,B 0,C 180,E1 -27764.655,E2 -27764.655} C_VEL
LIN {X 0,Y 94.586,Z 453.298,A -85,B 0,C 180,E1 -27768.031,E2 -27768.031} C_VEL
LIN {X 0,Y 88.942,Z 458.793,A -85,B 0,C 180,E1 -27773.656,E2 -27773.656} C_VEL
LIN {X 0,Y 84.16,Z 463.121,A -85,B 0,C 180,E1 -27779.931,E2 -27779.931} C_VEL
LIN {X 0,Y 81.523,Z 465.49,A -85,B 0,C 180,E1 -27784.466,E2 -27784.466} C_VEL
LIN {X 0,Y 79.549,Z 467.298,A -85,B 0,C 180,E1 -27789.305,E2 -27789.305} C_VEL
LIN {X 0,Y 77.14,Z 469.762,A -85,B 0,C 180,E1 -27799.501,E2 -27799.501} C_VEL
LIN {X 0,Y 76.735,Z 470.36,A -85,B 0,C 180,E1 -27804.745,E2 -27804.745} C_VEL
LIN {X 0,Y 76.781,Z 470.523,A -85,B 0,C 180,E1 -27810,E2 -27810} C_VEL
LIN {X 0,Y 76.711,Z 470.36,A -85,B 0,C 180,E1 -27815.257,E2 -27815.257} C_VEL
LIN {X 0,Y 77.125,Z 469.761,A -85,B 0,C 180,E1 -27820.501,E2 -27820.501} C_VEL
LIN {X 0,Y 79.549,Z 467.298,A -85,B 0,C 180,E1 -27830.695,E2 -27830.695} C_VEL
LIN {X 0,Y 82.782,Z 464.339,A -85,B 0,C 180,E1 -27837.836,E2 -27837.836} C_VEL
LIN {X 0,Y 87.23,Z 460.347,A -85,B 0,C 180,E1 -27844.331,E2 -27844.331} C_VEL
LIN {X 0,Y 92.69,Z 455.217,A -85,B 0,C 180,E1 -27850.128,E2 -27850.128} C_VEL
LIN {X 0,Y 97.625,Z 450.067,A -85,B 0,C 180,E1 -27854.435,E2 -27854.435} C_VEL
LIN {X 0,Y 102.167,Z 445.009,A -85,B 0,C 180,E1 -27857.687,E2 -27857.687} C_VEL
LIN {X 0,Y 103.18,Z 443.627,A -85,B 0,C 180,E1 -27858.526,E2 -27858.526} C_VEL
LIN {X 0,Y 106.024,Z 437.588,A -85,B 0,C 180,E1 -27862.697,E2 -27862.697} C_VEL
LIN {X 0,Y 107.982,Z 432.461,A -85,B 0,C 180,E1 -27866.106,E2 -27866.106} C_VEL
LIN {X 0,Y 109.142,Z 428.093,A -85,B 0,C 180,E1 -27868.991,E2 -27868.991} C_VEL
LIN {X 0,Y 109.456,Z 424.126,A -85,B 0,C 180,E1 -27872.254,E2 -27872.254} C_VEL
LIN {X 0,Y 109.299,Z 420.864,A -85,B 0,C 180,E1 -27875.29,E2 -27875.29} C_VEL
LIN {X 0,Y 108.944,Z 416.78,A -85,B 0,C 180,E1 -27879.823,E2 -27879.823} C_VEL
LIN {X 0,Y 108.638,Z 414.083,A -85,B 0,C 180,E1 -27883.073,E2 -27883.073} C_VEL
LIN {X 0,Y 108.038,Z 410.678,A -85,B 0,C 180,E1 -27888.744,E2 -27888.744} C_VEL
LIN {X 0,Y 107.401,Z 408.432,A -85,B 0,C 180,E1 -27896.246,E2 -27896.246} C_VEL
LIN {X 0,Y 107.725,Z 407.37,A -85,B 0,C 180,E1 -27899.998,E2 -27899.998} C_VEL
LIN {X 0,Y 107.628,Z 410.328,A -85,B 0,C 180,E1 -27911.627,E2 -27911.627} C_VEL
LIN {X 0,Y 108.353,Z 412.791,A -85,B 0,C 180,E1 -27916.968,E2 -27916.968} C_VEL
LIN {X 0,Y 109.33,Z 416.405,A -85,B 0,C 180,E1 -27922.685,E2 -27922.685} C_VEL
LIN {X 0,Y 109.987,Z 419.428,A -85,B 0,C 180,E1 -27926.567,E2 -27926.567} C_VEL
LIN {X 0,Y 110.821,Z 424.613,A -85,B 0,C 180,E1 -27932.156,E2 -27932.156} C_VEL
LIN {X 0,Y 111.281,Z 429.598,A -85,B 0,C 180,E1 -27936.866,E2 -27936.866} C_VEL
LIN {X 0,Y 111.12,Z 436.403,A -85,B 0,C 180,E1 -27942.883,E2 -27942.883} C_VEL
LIN {X 0,Y 110.426,Z 442.219,A -85,B 0,C 180,E1 -27948.069,E2 -27948.069} C_VEL
LIN {X 0,Y 109.635,Z 448.888,A -85,B 0,C 180,E1 -27954.765,E2 -27954.765} C_VEL
LIN {X 0,Y 110.473,Z 453.924,A -85,B 0,C 180,E1 -27961.203,E2 -27961.203} C_VEL
LIN {X 0,Y 112.201,Z 457.054,A -85,B 0,C 180,E1 -27965.975,E2 -27965.975} C_VEL
LIN {X 0,Y 117.254,Z 460.844,A -85,B 0,C 180,E1 -27973.532,E2 -27973.532} C_VEL
LIN {X 0,Y 122.316,Z 462.753,A -85,B 0,C 180,E1 -27978.472,E2 -27978.472} C_VEL
LIN {X 0,Y 123.706,Z 463.276,A -85,B 0,C 180,E1 -27980.202,E2 -27980.202} C_VEL
LIN {X 0,Y 124.624,Z 464.21,A -85,B 0,C 180,E1 -27983.271,E2 -27983.271} C_VEL
LIN {X 0,Y 125.95,Z 464.74,A -85,B 0,C 180,E1 -27986.276,E2 -27986.276} C_VEL
LIN {X 0,Y 127.895,Z 464.811,A -85,B 0,C 180,E1 -27987.836,E2 -27987.836} C_VEL
LIN {X 0,Y 132.192,Z 464.759,A -85,B 0,C 180,E1 -27990,E2 -27990} C_VEL
LIN {X 0,Y 126.003,Z 464.783,A -85,B 0,C 180,E1 -27993.197,E2 -27993.197} C_VEL
LIN {X 0,Y 120.306,Z 464.367,A -85,B 0,C 180,E1 -27996.752,E2 -27996.752} C_VEL
LIN {X 0,Y 114.637,Z 463.313,A -85,B 0,C 180,E1 -28001.225,E2 -28001.225} C_VEL
LIN {X 0,Y 107.887,Z 460.648,A -85,B 0,C 180,E1 -28009.009,E2 -28009.009} C_VEL
LIN {X 0,Y 104.406,Z 457.315,A -85,B 0,C 180,E1 -28015.908,E2 -28015.908} C_VEL
LIN {X 0,Y 102.945,Z 452.788,A -85,B 0,C 180,E1 -28023.103,E2 -28023.103} C_VEL
LIN {X 0,Y 103.26,Z 447.398,A -85,B 0,C 180,E1 -28029.834,E2 -28029.834} C_VEL
LIN {X 0,Y 104.4,Z 442.445,A -85,B 0,C 180,E1 -28034.978,E2 -28034.978} C_VEL
LIN {X 0,Y 105.195,Z 436.757,A -85,B 0,C 180,E1 -28040.606,E2 -28040.606} C_VEL
LIN {X 0,Y 105.428,Z 431.023,A -85,B 0,C 180,E1 -28046.373,E2 -28046.373} C_VEL
LIN {X 0,Y 105.234,Z 427.476,A -85,B 0,C 180,E1 -28050.25,E2 -28050.25} C_VEL
LIN {X 0,Y 104.89,Z 423.781,A -85,B 0,C 180,E1 -28054.856,E2 -28054.856} C_VEL
LIN {X 0,Y 104.275,Z 420.069,A -85,B 0,C 180,E1 -28060.309,E2 -28060.309} C_VEL
LIN {X 0,Y 103.885,Z 417.903,A -85,B 0,C 180,E1 -28064.302,E2 -28064.302} C_VEL
LIN {X 0,Y 103.575,Z 416.296,A -85,B 0,C 180,E1 -28068.257,E2 -28068.257} C_VEL
LIN {X 0,Y 103.354,Z 414.269,A -85,B 0,C 180,E1 -28076.103,E2 -28076.103} C_VEL
LIN {X 0,Y 103.781,Z 413.441,A -85,B 0,C 180,E1 -28080.002,E2 -28080.002} C_VEL
LIN {X 0,Y 103.661,Z 415.482,A -85,B 0,C 180,E1 -28087.795,E2 -28087.795} C_VEL
LIN {X 0,Y 103.98,Z 416.925,A -85,B 0,C 180,E1 -28091.701,E2 -28091.701} C_VEL
LIN {X 0,Y 104.112,Z 419.153,A -85,B 0,C 180,E1 -28095.667,E2 -28095.667} C_VEL
LIN {X 0,Y 104.286,Z 423.805,A -85,B 0,C 180,E1 -28101.758,E2 -28101.758} C_VEL
LIN {X 0,Y 104.166,Z 427.592,A -85,B 0,C 180,E1 -28105.866,E2 -28105.866} C_VEL
LIN {X 0,Y 103.89,Z 430.28,A -85,B 0,C 180,E1 -28108.427,E2 -28108.427} C_VEL
LIN {X 0,Y 102.784,Z 434.046,A -85,B 0,C 180,E1 -28111.274,E2 -28111.274} C_VEL
LIN {X 0,Y 99.839,Z 440.612,A -85,B 0,C 180,E1 -28115.951,E2 -28115.951} C_VEL
LIN {X 0,Y 97.467,Z 444.811,A -85,B 0,C 180,E1 -28119.182,E2 -28119.182} C_VEL
LIN {X 0,Y 90.524,Z 452.065,A -85,B 0,C 180,E1 -28124.099,E2 -28124.099} C_VEL
LIN {X 0,Y 85.325,Z 456.937,A -85,B 0,C 180,E1 -28128.781,E2 -28128.781} C_VEL
LIN {X 0,Y 79.72,Z 461.683,A -85,B 0,C 180,E1 -28135.038,E2 -28135.038} C_VEL
LIN {X 0,Y 75.149,Z 465.294,A -85,B 0,C 180,E1 -28142.121,E2 -28142.121} C_VEL
LIN {X 0,Y 72.917,Z 467.101,A -85,B 0,C 180,E1 -28147.323,E2 -28147.323} C_VEL
LIN {X 0,Y 70.158,Z 469.565,A -85,B 0,C 180,E1 -28158.443,E2 -28158.443} C_VEL
LIN {X 0,Y 69.648,Z 470.164,A -85,B 0,C 180,E1 -28164.209,E2 -28164.209} C_VEL
LIN {X 0,Y 69.701,Z 470.327,A -85,B 0,C 180,E1 -28170,E2 -28170} C_VEL
LIN {X 0,Y 69.624,Z 470.163,A -85,B 0,C 180,E1 -28175.793,E2 -28175.793} C_VEL
LIN {X 0,Y 70.146,Z 469.565,A -85,B 0,C 180,E1 -28181.559,E2 -28181.559} C_VEL
LIN {X 0,Y 72.917,Z 467.101,A -85,B 0,C 180,E1 -28192.677,E2 -28192.677} C_VEL
LIN {X 0,Y 76.555,Z 464.143,A -85,B 0,C 180,E1 -28200.326,E2 -28200.326} C_VEL
LIN {X 0,Y 81.432,Z 460.15,A -85,B 0,C 180,E1 -28207.167,E2 -28207.167} C_VEL
LIN {X 0,Y 86.772,Z 455.562,A -85,B 0,C 180,E1 -28212.61,E2 -28212.61} C_VEL
LIN {X 0,Y 92.765,Z 449.754,A -85,B 0,C 180,E1 -28217.618,E2 -28217.618} C_VEL
LIN {X 0,Y 97.446,Z 444.81,A -85,B 0,C 180,E1 -28220.833,E2 -28220.833} C_VEL
LIN {X 0,Y 100.773,Z 438.624,A -85,B 0,C 180,E1 -28225.451,E2 -28225.451} C_VEL
LIN {X 0,Y 102.756,Z 434.045,A -85,B 0,C 180,E1 -28228.753,E2 -28228.753} C_VEL
LIN {X 0,Y 103.89,Z 430.28,A -85,B 0,C 180,E1 -28231.573,E2 -28231.573} C_VEL
LIN {X 0,Y 104.292,Z 425.697,A -85,B 0,C 180,E1 -28236.149,E2 -28236.149} C_VEL
LIN {X 0,Y 104.184,Z 421.707,A -85,B 0,C 180,E1 -28240.804,E2 -28240.804} C_VEL
LIN {X 0,Y 104.137,Z 419.118,A -85,B 0,C 180,E1 -28244.336,E2 -28244.336} C_VEL
LIN {X 0,Y 104,Z 416.899,A -85,B 0,C 180,E1 -28248.301,E2 -28248.301} C_VEL
LIN {X 0,Y 103.679,Z 415.455,A -85,B 0,C 180,E1 -28252.206,E2 -28252.206} C_VEL
LIN {X 0,Y 103.816,Z 413.387,A -85,B 0,C 180,E1 -28259.998,E2 -28259.998} C_VEL
LIN {X 0,Y 103.341,Z 415.18,A -85,B 0,C 180,E1 -28267.815,E2 -28267.815} C_VEL
LIN {X 0,Y 103.567,Z 416.308,A -85,B 0,C 180,E1 -28271.744,E2 -28271.744} C_VEL
LIN {X 0,Y 103.867,Z 417.926,A -85,B 0,C 180,E1 -28275.701,E2 -28275.701} C_VEL
LIN {X 0,Y 104.541,Z 421.316,A -85,B 0,C 180,E1 -28281.698,E2 -28281.698} C_VEL
LIN {X 0,Y 104.989,Z 424.861,A -85,B 0,C 180,E1 -28286.573,E2 -28286.573} C_VEL
LIN {X 0,Y 105.429,Z 429.725,A -85,B 0,C 180,E1 -28292.225,E2 -28292.225} C_VEL
LIN {X 0,Y 105.376,Z 434.119,A -85,B 0,C 180,E1 -28296.885,E2 -28296.885} C_VEL
LIN {X 0,Y 104.864,Z 439.396,A -85,B 0,C 180,E1 -28302.08,E2 -28302.08} C_VEL
LIN {X 0,Y 103.871,Z 444.77,A -85,B 0,C 180,E1 -28307.421,E2 -28307.421} C_VEL
LIN {X 0,Y 102.882,Z 450.509,A -85,B 0,C 180,E1 -28313.921,E2 -28313.921} C_VEL
LIN {X 0,Y 103.209,Z 454.369,A -85,B 0,C 180,E1 -28319.289,E2 -28319.289} C_VEL
LIN {X 0,Y 104.38,Z 457.316,A -85,B 0,C 180,E1 -28324.085,E2 -28324.085} C_VEL
LIN {X 0,Y 107.856,Z 460.649,A -85,B 0,C 180,E1 -28330.986,E2 -28330.986} C_VEL
LIN {X 0,Y 114.638,Z 463.313,A -85,B 0,C 180,E1 -28338.773,E2 -28338.773} C_VEL
LIN {X 0,Y 120.384,Z 464.372,A -85,B 0,C 180,E1 -28343.295,E2 -28343.295} C_VEL
LIN {X 0,Y 127.895,Z 464.811,A -85,B 0,C 180,E1 -28347.836,E2 -28347.836} C_VEL
LIN {X 0,Y 128.328,Z 464.866,A -85,B 0,C 180,E1 -28348.603,E2 -28348.603} C_VEL
LIN {X 0,Y 127.523,Z 464.887,A -85,B 0,C 180,E1 -28349.644,E2 -28349.644} C_VEL
LIN {X 0,Y 125.058,Z 464.966,A -85,B 0,C 180,E1 -28350.962,E2 -28350.962} C_VEL
LIN {X 0,Y 115.293,Z 464.934,A -85,B 0,C 180,E1 -28354.428,E2 -28354.428} C_VEL
LIN {X 0,Y 113.664,Z 464.831,A -85,B 0,C 180,E1 -28355.373,E2 -28355.373} C_VEL
LIN {X 0,Y 106.482,Z 463.742,A -85,B 0,C 180,E1 -28361.42,E2 -28361.42} C_VEL
LIN {X 0,Y 102.421,Z 462.444,A -85,B 0,C 180,E1 -28366.132,E2 -28366.132} C_VEL
LIN {X 0,Y 98.762,Z 460.191,A -85,B 0,C 180,E1 -28372.325,E2 -28372.325} C_VEL
LIN {X 0,Y 96.318,Z 456.076,A -85,B 0,C 180,E1 -28380.715,E2 -28380.715} C_VEL
LIN {X 0,Y 96.238,Z 451.183,A -85,B 0,C 180,E1 -28388.367,E2 -28388.367} C_VEL
LIN {X 0,Y 97.939,Z 444.998,A -85,B 0,C 180,E1 -28395.856,E2 -28395.856} C_VEL
LIN {X 0,Y 98.993,Z 440.037,A -85,B 0,C 180,E1 -28401.347,E2 -28401.347} C_VEL
LIN {X 0,Y 99.54,Z 436.287,A -85,B 0,C 180,E1 -28405.612,E2 -28405.612} C_VEL
LIN {X 0,Y 99.746,Z 432.211,A -85,B 0,C 180,E1 -28410.451,E2 -28410.451} C_VEL
LIN {X 0,Y 99.617,Z 427.821,A -85,B 0,C 180,E1 -28416.513,E2 -28416.513} C_VEL
LIN {X 0,Y 99.45,Z 425.087,A -85,B 0,C 180,E1 -28421.053,E2 -28421.053} C_VEL
LIN {X 0,Y 99.142,Z 422.134,A -85,B 0,C 180,E1 -28427.724,E2 -28427.724} C_VEL
LIN {X 0,Y 98.982,Z 420.464,A -85,B 0,C 180,E1 -28433.736,E2 -28433.736} C_VEL
LIN {X 0,Y 99.569,Z 419.246,A -85,B 0,C 180,E1 -28440.002,E2 -28440.002} C_VEL
LIN {X 0,Y 99.297,Z 421.272,A -85,B 0,C 180,E1 -28448.14,E2 -28448.14} C_VEL
LIN {X 0,Y 99.434,Z 422.914,A -85,B 0,C 180,E1 -28452.244,E2 -28452.244} C_VEL
LIN {X 0,Y 99.37,Z 425.394,A -85,B 0,C 180,E1 -28456.436,E2 -28456.436} C_VEL
LIN {X 0,Y 99.163,Z 428.402,A -85,B 0,C 180,E1 -28460.757,E2 -28460.757} C_VEL
LIN {X 0,Y 98.746,Z 432.334,A -85,B 0,C 180,E1 -28465.282,E2 -28465.282} C_VEL
LIN {X 0,Y 98.216,Z 434.339,A -85,B 0,C 180,E1 -28467.291,E2 -28467.291} C_VEL
LIN {X 0,Y 96.274,Z 438.633,A -85,B 0,C 180,E1 -28470.733,E2 -28470.733} C_VEL
LIN {X 0,Y 92.763,Z 444.597,A -85,B 0,C 180,E1 -28475.467,E2 -28475.467} C_VEL
LIN {X 0,Y 91.876,Z 445.992,A -85,B 0,C 180,E1 -28476.565,E2 -28476.565} C_VEL
LIN {X 0,Y 83.574,Z 453.679,A -85,B 0,C 180,E1 -28482.283,E2 -28482.283} C_VEL
LIN {X 0,Y 77.939,Z 458.4,A -85,B 0,C 180,E1 -28487.445,E2 -28487.445} C_VEL
LIN {X 0,Y 72.183,Z 462.728,A -85,B 0,C 180,E1 -28494.255,E2 -28494.255} C_VEL
LIN {X 0,Y 68.931,Z 465.097,A -85,B 0,C 180,E1 -28499.35,E2 -28499.35} C_VEL
LIN {X 0,Y 66.375,Z 466.904,A -85,B 0,C 180,E1 -28504.942,E2 -28504.942} C_VEL
LIN {X 0,Y 63.192,Z 469.369,A -85,B 0,C 180,E1 -28517.148,E2 -28517.148} C_VEL
LIN {X 0,Y 62.578,Z 469.968,A -85,B 0,C 180,E1 -28523.552,E2 -28523.552} C_VEL
LIN {X 0,Y 62.611,Z 470.132,A -85,B 0,C 180,E1 -28530,E2 -28530} C_VEL
LIN {X 0,Y 62.559,Z 469.967,A -85,B 0,C 180,E1 -28536.45,E2 -28536.45} C_VEL
LIN {X 0,Y 63.183,Z 469.369,A -85,B 0,C 180,E1 -28542.854,E2 -28542.854} C_VEL
LIN {X 0,Y 66.376,Z 466.904,A -85,B 0,C 180,E1 -28555.057,E2 -28555.057} C_VEL
LIN {X 0,Y 70.503,Z 463.946,A -85,B 0,C 180,E1 -28563.248,E2 -28563.248} C_VEL
LIN {X 0,Y 75.871,Z 459.953,A -85,B 0,C 180,E1 -28570.422,E2 -28570.422} C_VEL
LIN {X 0,Y 81.358,Z 455.625,A -85,B 0,C 180,E1 -28575.741,E2 -28575.741} C_VEL
LIN {X 0,Y 86.913,Z 450.714,A -85,B 0,C 180,E1 -28580.191,E2 -28580.191} C_VEL
LIN {X 0,Y 91.856,Z 445.991,A -85,B 0,C 180,E1 -28583.452,E2 -28583.452} C_VEL
LIN {X 0,Y 95.656,Z 439.884,A -85,B 0,C 180,E1 -28588.33,E2 -28588.33} C_VEL
LIN {X 0,Y 98.228,Z 434.318,A -85,B 0,C 180,E1 -28592.722,E2 -28592.722} C_VEL
LIN {X 0,Y 98.878,Z 431.131,A -85,B 0,C 180,E1 -28596.026,E2 -28596.026} C_VEL
LIN {X 0,Y 99.258,Z 427.044,A -85,B 0,C 180,E1 -28601.085,E2 -28601.085} C_VEL
LIN {X 0,Y 99.488,Z 424.007,A -85,B 0,C 180,E1 -28605.683,E2 -28605.683} C_VEL
LIN {X 0,Y 99.45,Z 422.893,A -85,B 0,C 180,E1 -28607.758,E2 -28607.758} C_VEL
LIN {X 0,Y 99.315,Z 421.135,A -85,B 0,C 180,E1 -28612.182,E2 -28612.182} C_VEL
LIN {X 0,Y 99.6,Z 419.205,A -85,B 0,C 180,E1 -28619.998,E2 -28619.998} C_VEL
LIN {X 0,Y 98.969,Z 420.922,A -85,B 0,C 180,E1 -28628.163,E2 -28628.163} C_VEL
LIN {X 0,Y 99.115,Z 422.169,A -85,B 0,C 180,E1 -28632.28,E2 -28632.28} C_VEL
LIN {X 0,Y 99.452,Z 425.075,A -85,B 0,C 180,E1 -28638.929,E2 -28638.929} C_VEL
LIN {X 0,Y 99.688,Z 428.876,A -85,B 0,C 180,E1 -28645.022,E2 -28645.022} C_VEL
LIN {X 0,Y 99.731,Z 433.241,A -85,B 0,C 180,E1 -28650.877,E2 -28650.877} C_VEL
LIN {X 0,Y 99.448,Z 437.537,A -85,B 0,C 180,E1 -28655.819,E2 -28655.819} C_VEL
LIN {X 0,Y 98.459,Z 443.017,A -85,B 0,C 180,E1 -28661.855,E2 -28661.855} C_VEL
LIN {X 0,Y 97.203,Z 447.488,A -85,B 0,C 180,E1 -28666.949,E2 -28666.949} C_VEL
LIN {X 0,Y 96.083,Z 453.018,A -85,B 0,C 180,E1 -28674.186,E2 -28674.186} C_VEL
LIN {X 0,Y 96.588,Z 456.959,A -85,B 0,C 180,E1 -28680.822,E2 -28680.822} C_VEL
LIN {X 0,Y 99.586,Z 460.891,A -85,B 0,C 180,E1 -28689.338,E2 -28689.338} C_VEL
LIN {X 0,Y 102.572,Z 462.524,A -85,B 0,C 180,E1 -28694.093,E2 -28694.093} C_VEL
LIN {X 0,Y 111.151,Z 464.628,A -85,B 0,C 180,E1 -28702.735,E2 -28702.735} C_VEL
LIN {X 0,Y 119.524,Z 465.109,A -85,B 0,C 180,E1 -28708.311,E2 -28708.311} C_VEL
LIN {X 0,Y 122.632,Z 465.022,A -85,B 0,C 180,E1 -28710,E2 -28710} C_VEL
LIN {X 0,Y 113.664,Z 464.831,A -85,B 0,C 180,E1 -28715.373,E2 -28715.373} C_VEL
LIN {X 0,Y 109.807,Z 464.617,A -85,B 0,C 180,E1 -28717.673,E2 -28717.673} C_VEL
LIN {X 0,Y 97.162,Z 463.48,A -85,B 0,C 180,E1 -28724.618,E2 -28724.618} C_VEL
LIN {X 0,Y 94.087,Z 462.699,A -85,B 0,C 180,E1 -28727.58,E2 -28727.58} C_VEL
LIN {X 0,Y 93.374,Z 462.352,A -85,B 0,C 180,E1 -28728.675,E2 -28728.675} C_VEL
LIN {X 0,Y 90.519,Z 460.063,A -85,B 0,C 180,E1 -28735.276,E2 -28735.276} C_VEL
LIN {X 0,Y 89.22,Z 456.307,A -85,B 0,C 180,E1 -28743.463,E2 -28743.463} C_VEL
LIN {X 0,Y 89.498,Z 453.246,A -85,B 0,C 180,E1 -28748.918,E2 -28748.918} C_VEL
LIN {X 0,Y 91.626,Z 447.012,A -85,B 0,C 180,E1 -28757.417,E2 -28757.417} C_VEL
LIN {X 0,Y 92.896,Z 442.807,A -85,B 0,C 180,E1 -28762.757,E2 -28762.757} C_VEL
LIN {X 0,Y 93.8,Z 438.391,A -85,B 0,C 180,E1 -28768.37,E2 -28768.37} C_VEL
LIN {X 0,Y 94.158,Z 434.661,A -85,B 0,C 180,E1 -28773.596,E2 -28773.596} C_VEL
LIN {X 0,Y 94.452,Z 430.597,A -85,B 0,C 180,E1 -28780.44,E2 -28780.44} C_VEL
LIN {X 0,Y 94.313,Z 427.722,A -85,B 0,C 180,E1 -28787.085,E2 -28787.085} C_VEL
LIN {X 0,Y 94.308,Z 426.469,A -85,B 0,C 180,E1 -28791.431,E2 -28791.431} C_VEL
LIN {X 0,Y 95.101,Z 424.846,A -85,B 0,C 180,E1 -28800.002,E2 -28800.002} C_VEL
LIN {X 0,Y 94.616,Z 426.906,A -85,B 0,C 180,E1 -28808.546,E2 -28808.546} C_VEL
LIN {X 0,Y 94.54,Z 428.632,A -85,B 0,C 180,E1 -28812.889,E2 -28812.889} C_VEL
LIN {X 0,Y 93.946,Z 432.875,A -85,B 0,C 180,E1 -28819.675,E2 -28819.675} C_VEL
LIN {X 0,Y 93.228,Z 435.877,A -85,B 0,C 180,E1 -28823.665,E2 -28823.665} C_VEL
LIN {X 0,Y 92.623,Z 437.576,A -85,B 0,C 180,E1 -28825.474,E2 -28825.474} C_VEL
LIN {X 0,Y 90.722,Z 441.03,A -85,B 0,C 180,E1 -28828.469,E2 -28828.469} C_VEL
LIN {X 0,Y 87.49,Z 445.778,A -85,B 0,C 180,E1 -28832.494,E2 -28832.494} C_VEL
LIN {X 0,Y 86.478,Z 447.049,A -85,B 0,C 180,E1 -28833.591,E2 -28833.591} C_VEL
LIN {X 0,Y 79.978,Z 452.708,A -85,B 0,C 180,E1 -28837.734,E2 -28837.734} C_VEL
LIN {X 0,Y 72.856,Z 458.204,A -85,B 0,C 180,E1 -28843.657,E2 -28843.657} C_VEL
LIN {X 0,Y 66.536,Z 462.532,A -85,B 0,C 180,E1 -28850.672,E2 -28850.672} C_VEL
LIN {X 0,Y 62.911,Z 464.901,A -85,B 0,C 180,E1 -28856.043,E2 -28856.043} C_VEL
LIN {X 0,Y 57.774,Z 468.104,A -85,B 0,C 180,E1 -28868.596,E2 -28868.596} C_VEL
LIN {X 0,Y 56.279,Z 469.173,A -85,B 0,C 180,E1 -28875.537,E2 -28875.537} C_VEL
LIN {X 0,Y 55.531,Z 469.772,A -85,B 0,C 180,E1 -28882.729,E2 -28882.729} C_VEL
LIN {X 0,Y 55.509,Z 469.936,A -85,B 0,C 180,E1 -28890,E2 -28890} C_VEL
LIN {X 0,Y 55.517,Z 469.772,A -85,B 0,C 180,E1 -28897.273,E2 -28897.273} C_VEL
LIN {X 0,Y 56.271,Z 469.172,A -85,B 0,C 180,E1 -28904.465,E2 -28904.465} C_VEL
LIN {X 0,Y 59.977,Z 466.707,A -85,B 0,C 180,E1 -28917.951,E2 -28917.951} C_VEL
LIN {X 0,Y 64.671,Z 463.75,A -85,B 0,C 180,E1 -28926.705,E2 -28926.705} C_VEL
LIN {X 0,Y 70.599,Z 459.757,A -85,B 0,C 180,E1 -28934.173,E2 -28934.173} C_VEL
LIN {X 0,Y 77.25,Z 454.83,A -85,B 0,C 180,E1 -28940.213,E2 -28940.213} C_VEL
LIN {X 0,Y 83.812,Z 449.36,A -85,B 0,C 180,E1 -28944.843,E2 -28944.843} C_VEL
LIN {X 0,Y 86.449,Z 447.048,A -85,B 0,C 180,E1 -28946.437,E2 -28946.437} C_VEL
LIN {X 0,Y 89.393,Z 442.98,A -85,B 0,C 180,E1 -28949.86,E2 -28949.86} C_VEL
LIN {X 0,Y 92.304,Z 438.234,A -85,B 0,C 180,E1 -28953.948,E2 -28953.948} C_VEL
LIN {X 0,Y 93.228,Z 435.877,A -85,B 0,C 180,E1 -28956.334,E2 -28956.334} C_VEL
LIN {X 0,Y 93.911,Z 432.911,A -85,B 0,C 180,E1 -28960.318,E2 -28960.318} C_VEL
LIN {X 0,Y 94.416,Z 429.573,A -85,B 0,C 180,E1 -28965.39,E2 -28965.39} C_VEL
LIN {X 0,Y 94.564,Z 428.606,A -85,B 0,C 180,E1 -28967.115,E2 -28967.115} C_VEL
LIN {X 0,Y 94.626,Z 426.895,A -85,B 0,C 180,E1 -28971.455,E2 -28971.455} C_VEL
LIN {X 0,Y 95.131,Z 424.814,A -85,B 0,C 180,E1 -28979.998,E2 -28979.998} C_VEL
LIN {X 0,Y 94.295,Z 426.483,A -85,B 0,C 180,E1 -28988.57,E2 -28988.57} C_VEL
LIN {X 0,Y 94.286,Z 428.274,A -85,B 0,C 180,E1 -28994.303,E2 -28994.303} C_VEL
LIN {X 0,Y 94.43,Z 430.62,A -85,B 0,C 180,E1 -28999.565,E2 -28999.565} C_VEL
LIN {X 0,Y 94.158,Z 434.661,A -85,B 0,C 180,E1 -29006.403,E2 -29006.403} C_VEL
LIN {X 0,Y 93.821,Z 438.371,A -85,B 0,C 180,E1 -29011.622,E2 -29011.622} C_VEL
LIN {X 0,Y 92.906,Z 442.798,A -85,B 0,C 180,E1 -29017.238,E2 -29017.238} C_VEL
LIN {X 0,Y 91.6,Z 447.016,A -85,B 0,C 180,E1 -29022.57,E2 -29022.57} C_VEL
LIN {X 0,Y 89.969,Z 451.407,A -85,B 0,C 180,E1 -29028.396,E2 -29028.396} C_VEL
LIN {X 0,Y 89.228,Z 455.014,A -85,B 0,C 180,E1 -29034.139,E2 -29034.139} C_VEL
LIN {X 0,Y 89.849,Z 458.924,A -85,B 0,C 180,E1 -29042.01,E2 -29042.01} C_VEL
LIN {X 0,Y 91.479,Z 461.132,A -85,B 0,C 180,E1 -29047.41,E2 -29047.41} C_VEL
LIN {X 0,Y 95.013,Z 463.227,A -85,B 0,C 180,E1 -29054.06,E2 -29054.06} C_VEL
LIN {X 0,Y 102.041,Z 464.882,A -85,B 0,C 180,E1 -29062.082,E2 -29062.082} C_VEL
LIN {X 0,Y 107.182,Z 465.303,A -85,B 0,C 180,E1 -29066.24,E2 -29066.24} C_VEL
LIN {X 0,Y 113.126,Z 465.284,A -85,B 0,C 180,E1 -29070,E2 -29070} C_VEL
LIN {X 0,Y 105.783,Z 465.197,A -85,B 0,C 180,E1 -29074.775,E2 -29074.775} C_VEL
LIN {X 0,Y 99.899,Z 464.537,A -85,B 0,C 180,E1 -29079.98,E2 -29079.98} C_VEL
LIN {X 0,Y 94.116,Z 462.768,A -85,B 0,C 180,E1 -29087.379,E2 -29087.379} C_VEL
LIN {X 0,Y 93.374,Z 462.352,A -85,B 0,C 180,E1 -29088.675,E2 -29088.675} C_VEL
LIN {X 0,Y 91.087,Z 461.401,A -85,B 0,C 180,E1 -29092.011,E2 -29092.011} C_VEL
LIN {X 0,Y 83.46,Z 458.286,A -85,B 0,C 180,E1 -29102.413,E2 -29102.413} C_VEL
LIN {X 0,Y 82.454,Z 456.721,A -85,B 0,C 180,E1 -29106.257,E2 -29106.257} C_VEL
LIN {X 0,Y 82.478,Z 456.089,A -85,B 0,C 180,E1 -29107.546,E2 -29107.546} C_VEL
LIN {X 0,Y 84.079,Z 451.63,A -85,B 0,C 180,E1 -29115.275,E2 -29115.275} C_VEL
LIN {X 0,Y 85.253,Z 449.339,A -85,B 0,C 180,E1 -29118.742,E2 -29118.742} C_VEL
LIN {X 0,Y 87.04,Z 444.523,A -85,B 0,C 180,E1 -29125.586,E2 -29125.586} C_VEL
LIN {X 0,Y 88.083,Z 440.558,A -85,B 0,C 180,E1 -29131.4,E2 -29131.4} C_VEL
LIN {X 0,Y 88.7,Z 437.5,A -85,B 0,C 180,E1 -29136.664,E2 -29136.664} C_VEL
LIN {X 0,Y 89.073,Z 434.869,A -85,B 0,C 180,E1 -29141.605,E2 -29141.605} C_VEL
LIN {X 0,Y 89.21,Z 433.069,A -85,B 0,C 180,E1 -29146.332,E2 -29146.332} C_VEL
LIN {X 0,Y 89.363,Z 431.814,A -85,B 0,C 180,E1 -29150.953,E2 -29150.953} C_VEL
LIN {X 0,Y 90.239,Z 430.141,A -85,B 0,C 180,E1 -29160.002,E2 -29160.002} C_VEL
LIN {X 0,Y 89.824,Z 431.087,A -85,B 0,C 180,E1 -29164.49,E2 -29164.49} C_VEL
LIN {X 0,Y 89.621,Z 432.342,A -85,B 0,C 180,E1 -29169.026,E2 -29169.026} C_VEL
LIN {X 0,Y 89.184,Z 434.258,A -85,B 0,C 180,E1 -29173.677,E2 -29173.677} C_VEL
LIN {X 0,Y 88.45,Z 437.027,A -85,B 0,C 180,E1 -29178.534,E2 -29178.534} C_VEL
LIN {X 0,Y 87.56,Z 439.814,A -85,B 0,C 180,E1 -29182.414,E2 -29182.414} C_VEL
LIN {X 0,Y 86.761,Z 441.139,A -85,B 0,C 180,E1 -29183.895,E2 -29183.895} C_VEL
LIN {X 0,Y 83.532,Z 445.562,A -85,B 0,C 180,E1 -29187.943,E2 -29187.943} C_VEL
LIN {X 0,Y 81.324,Z 448.008,A -85,B 0,C 180,E1 -29190.209,E2 -29190.209} C_VEL
LIN {X 0,Y 75.817,Z 452.511,A -85,B 0,C 180,E1 -29193.461,E2 -29193.461} C_VEL
LIN {X 0,Y 68.136,Z 458.008,A -85,B 0,C 180,E1 -29199.322,E2 -29199.322} C_VEL
LIN {X 0,Y 61.196,Z 462.335,A -85,B 0,C 180,E1 -29206.444,E2 -29206.444} C_VEL
LIN {X 0,Y 57.149,Z 464.705,A -85,B 0,C 180,E1 -29212.057,E2 -29212.057} C_VEL
LIN {X 0,Y 53.77,Z 466.51,A -85,B 0,C 180,E1 -29218.478,E2 -29218.478} C_VEL
LIN {X 0,Y 49.402,Z 468.976,A -85,B 0,C 180,E1 -29233.47,E2 -29233.47} C_VEL
LIN {X 0,Y 48.489,Z 469.576,A -85,B 0,C 180,E1 -29241.666,E2 -29241.666} C_VEL
LIN {X 0,Y 48.427,Z 469.741,A -85,B 0,C 180,E1 -29250,E2 -29250} C_VEL
LIN {X 0,Y 48.477,Z 469.576,A -85,B 0,C 180,E1 -29258.336,E2 -29258.336} C_VEL
LIN {X 0,Y 49.396,Z 468.976,A -85,B 0,C 180,E1 -29266.532,E2 -29266.532} C_VEL
LIN {X 0,Y 53.77,Z 466.51,A -85,B 0,C 180,E1 -29281.522,E2 -29281.522} C_VEL
LIN {X 0,Y 59.101,Z 463.553,A -85,B 0,C 180,E1 -29290.846,E2 -29290.846} C_VEL
LIN {X 0,Y 65.681,Z 459.561,A -85,B 0,C 180,E1 -29298.504,E2 -29298.504} C_VEL
LIN {X 0,Y 72.182,Z 455.151,A -85,B 0,C 180,E1 -29304.02,E2 -29304.02} C_VEL
LIN {X 0,Y 79.914,Z 449.163,A -85,B 0,C 180,E1 -29309.031,E2 -29309.031} C_VEL
LIN {X 0,Y 81.318,Z 448.008,A -85,B 0,C 180,E1 -29309.798,E2 -29309.798} C_VEL
LIN {X 0,Y 83.522,Z 445.561,A -85,B 0,C 180,E1 -29312.07,E2 -29312.07} C_VEL
LIN {X 0,Y 86.729,Z 441.167,A -85,B 0,C 180,E1 -29316.095,E2 -29316.095} C_VEL
LIN {X 0,Y 87.532,Z 439.84,A -85,B 0,C 180,E1 -29317.578,E2 -29317.578} C_VEL
LIN {X 0,Y 88.551,Z 436.561,A -85,B 0,C 180,E1 -29322.249,E2 -29322.249} C_VEL
LIN {X 0,Y 89.242,Z 434.203,A -85,B 0,C 180,E1 -29326.332,E2 -29326.332} C_VEL
LIN {X 0,Y 89.633,Z 432.331,A -85,B 0,C 180,E1 -29330.975,E2 -29330.975} C_VEL
LIN {X 0,Y 90.279,Z 430.097,A -85,B 0,C 180,E1 -29339.998,E2 -29339.998} C_VEL
LIN {X 0,Y 89.336,Z 431.84,A -85,B 0,C 180,E1 -29349.05,E2 -29349.05} C_VEL
LIN {X 0,Y 89.187,Z 433.09,A -85,B 0,C 180,E1 -29353.672,E2 -29353.672} C_VEL
LIN {X 0,Y 89.035,Z 435.029,A -85,B 0,C 180,E1 -29358.698,E2 -29358.698} C_VEL
LIN {X 0,Y 88.7,Z 437.501,A -85,B 0,C 180,E1 -29363.336,E2 -29363.336} C_VEL
LIN {X 0,Y 88.101,Z 440.577,A -85,B 0,C 180,E1 -29368.659,E2 -29368.659} C_VEL
LIN {X 0,Y 87.058,Z 444.509,A -85,B 0,C 180,E1 -29374.405,E2 -29374.405} C_VEL
LIN {X 0,Y 85.89,Z 447.691,A -85,B 0,C 180,E1 -29378.987,E2 -29378.987} C_VEL
LIN {X 0,Y 84.093,Z 451.63,A -85,B 0,C 180,E1 -29384.734,E2 -29384.734} C_VEL
LIN {X 0,Y 82.391,Z 456.537,A -85,B 0,C 180,E1 -29393.338,E2 -29393.338} C_VEL
LIN {X 0,Y 82.916,Z 460.297,A -85,B 0,C 180,E1 -29402.213,E2 -29402.213} C_VEL
LIN {X 0,Y 85.751,Z 463.011,A -85,B 0,C 180,E1 -29410.863,E2 -29410.863} C_VEL
LIN {X 0,Y 92.545,Z 465.09,A -85,B 0,C 180,E1 -29420.822,E2 -29420.822} C_VEL
LIN {X 0,Y 98.584,Z 465.606,A -85,B 0,C 180,E1 -29426.382,E2 -29426.382} C_VEL
LIN {X 0,Y 103.691,Z 465.545,A -85,B 0,C 180,E1 -29430,E2 -29430} C_VEL
LIN {X 0,Y 97.965,Z 465.557,A -85,B 0,C 180,E1 -29434.114,E2 -29434.114} C_VEL
LIN {X 0,Y 92.548,Z 465.088,A -85,B 0,C 180,E1 -29439.19,E2 -29439.19} C_VEL
LIN {X 0,Y 85.761,Z 463.01,A -85,B 0,C 180,E1 -29449.135,E2 -29449.135} C_VEL
LIN {X 0,Y 82.932,Z 460.296,A -85,B 0,C 180,E1 -29457.781,E2 -29457.781} C_VEL
LIN {X 0,Y 82.398,Z 456.537,A -85,B 0,C 180,E1 -29466.659,E2 -29466.659} C_VEL
LIN {X 0,Y 82.478,Z 456.089,A -85,B 0,C 180,E1 -29467.546,E2 -29467.546} C_VEL
LIN {X 0,Y 82.486,Z 454.277,A -85,B 0,C 180,E1 -29471.449,E2 -29471.449} C_VEL
LIN {X 0,Y 81.57,Z 451.299,A -85,B 0,C 180,E1 -29478.044,E2 -29478.044} C_VEL
LIN {X 0,Y 80.968,Z 447.65,A -85,B 0,C 180,E1 -29486.135,E2 -29486.135} C_VEL
LIN {X 0,Y 81.332,Z 446.194,A -85,B 0,C 180,E1 -29488.775,E2 -29488.775} C_VEL
LIN {X 0,Y 82.543,Z 442.813,A -85,B 0,C 180,E1 -29494.807,E2 -29494.807} C_VEL
LIN {X 0,Y 83.273,Z 440.126,A -85,B 0,C 180,E1 -29500.273,E2 -29500.273} C_VEL
LIN {X 0,Y 83.742,Z 438.228,A -85,B 0,C 180,E1 -29505.42,E2 -29505.42} C_VEL
LIN {X 0,Y 84.018,Z 436.814,A -85,B 0,C 180,E1 -29510.372,E2 -29510.372} C_VEL
LIN {X 0,Y 84.522,Z 435.661,A -85,B 0,C 180,E1 -29516.198,E2 -29516.198} C_VEL
LIN {X 0,Y 85.076,Z 435.133,A -85,B 0,C 180,E1 -29520.003,E2 -29520.003} C_VEL
LIN {X 0,Y 84.561,Z 436.072,A -85,B 0,C 180,E1 -29524.77,E2 -29524.77} C_VEL
LIN {X 0,Y 84.127,Z 437.488,A -85,B 0,C 180,E1 -29529.621,E2 -29529.621} C_VEL
LIN {X 0,Y 83.882,Z 438.436,A -85,B 0,C 180,E1 -29532.093,E2 -29532.093} C_VEL
LIN {X 0,Y 82.794,Z 441.119,A -85,B 0,C 180,E1 -29537.448,E2 -29537.448} C_VEL
LIN {X 0,Y 82.041,Z 442.701,A -85,B 0,C 180,E1 -29540.042,E2 -29540.042} C_VEL
LIN {X 0,Y 80.071,Z 445.339,A -85,B 0,C 180,E1 -29542.839,E2 -29542.839} C_VEL
LIN {X 0,Y 77.754,Z 447.797,A -85,B 0,C 180,E1 -29545.328,E2 -29545.328} C_VEL
LIN {X 0,Y 76.497,Z 448.967,A -85,B 0,C 180,E1 -29546.395,E2 -29546.395} C_VEL
LIN {X 0,Y 68.843,Z 454.525,A -85,B 0,C 180,E1 -29550.696,E2 -29550.696} C_VEL
LIN {X 0,Y 61.199,Z 459.364,A -85,B 0,C 180,E1 -29556.499,E2 -29556.499} C_VEL
LIN {X 0,Y 53.909,Z 463.356,A -85,B 0,C 180,E1 -29564.191,E2 -29564.191} C_VEL
LIN {X 0,Y 47.828,Z 466.313,A -85,B 0,C 180,E1 -29574.001,E2 -29574.001} C_VEL
LIN {X 0,Y 42.62,Z 468.779,A -85,B 0,C 180,E1 -29590.743,E2 -29590.743} C_VEL
LIN {X 0,Y 41.46,Z 469.38,A -85,B 0,C 180,E1 -29600.241,E2 -29600.241} C_VEL
LIN {X 0,Y 41.326,Z 469.545,A -85,B 0,C 180,E1 -29610,E2 -29610} C_VEL
LIN {X 0,Y 41.451,Z 469.379,A -85,B 0,C 180,E1 -29619.762,E2 -29619.762} C_VEL
LIN {X 0,Y 42.615,Z 468.779,A -85,B 0,C 180,E1 -29629.259,E2 -29629.259} C_VEL
LIN {X 0,Y 47.828,Z 466.313,A -85,B 0,C 180,E1 -29645.999,E2 -29645.999} C_VEL
LIN {X 0,Y 53.909,Z 463.356,A -85,B 0,C 180,E1 -29655.809,E2 -29655.809} C_VEL
LIN {X 0,Y 61.2,Z 459.364,A -85,B 0,C 180,E1 -29663.5,E2 -29663.5} C_VEL
LIN {X 0,Y 69.277,Z 454.252,A -85,B 0,C 180,E1 -29669.516,E2 -29669.516} C_VEL
LIN {X 0,Y 76.488,Z 448.966,A -85,B 0,C 180,E1 -29673.619,E2 -29673.619} C_VEL
LIN {X 0,Y 78.909,Z 446.618,A -85,B 0,C 180,E1 -29675.91,E2 -29675.91} C_VEL
LIN {X 0,Y 81.2,Z 443.9,A -85,B 0,C 180,E1 -29678.576,E2 -29678.576} C_VEL
LIN {X 0,Y 82.127,Z 442.507,A -85,B 0,C 180,E1 -29680.274,E2 -29680.274} C_VEL
LIN {X 0,Y 83.441,Z 439.649,A -85,B 0,C 180,E1 -29685.361,E2 -29685.361} C_VEL
LIN {X 0,Y 83.919,Z 438.401,A -85,B 0,C 180,E1 -29687.912,E2 -29687.912} C_VEL
LIN {X 0,Y 84.158,Z 437.459,A -85,B 0,C 180,E1 -29690.383,E2 -29690.383} C_VEL
LIN {X 0,Y 84.584,Z 435.995,A -85,B 0,C 180,E1 -29695.606,E2 -29695.606} C_VEL
LIN {X 0,Y 85.1,Z 435.111,A -85,B 0,C 180,E1 -29699.997,E2 -29699.997} C_VEL
LIN {X 0,Y 83.984,Z 436.845,A -85,B 0,C 180,E1 -29709.632,E2 -29709.632} C_VEL
LIN {X 0,Y 83.728,Z 438.24,A -85,B 0,C 180,E1 -29714.582,E2 -29714.582} C_VEL
LIN {X 0,Y 83.271,Z 440.128,A -85,B 0,C 180,E1 -29719.728,E2 -29719.728} C_VEL
LIN {X 0,Y 82.508,Z 442.843,A -85,B 0,C 180,E1 -29725.204,E2 -29725.204} C_VEL
LIN {X 0,Y 81.359,Z 446.174,A -85,B 0,C 180,E1 -29731.215,E2 -29731.215} C_VEL
LIN {X 0,Y 79.596,Z 450.025,A -85,B 0,C 180,E1 -29737.377,E2 -29737.377} C_VEL
LIN {X 0,Y 76.79,Z 454.93,A -85,B 0,C 180,E1 -29745.787,E2 -29745.787} C_VEL
LIN {X 0,Y 75.562,Z 458.221,A -85,B 0,C 180,E1 -29752.803,E2 -29752.803} C_VEL
LIN {X 0,Y 75.96,Z 461.604,A -85,B 0,C 180,E1 -29762.444,E2 -29762.444} C_VEL
LIN {X 0,Y 77.57,Z 463.251,A -85,B 0,C 180,E1 -29768.752,E2 -29768.752} C_VEL
LIN {X 0,Y 84.114,Z 465.382,A -85,B 0,C 180,E1 -29780.38,E2 -29780.38} C_VEL
LIN {X 0,Y 91.431,Z 465.885,A -85,B 0,C 180,E1 -29787.74,E2 -29787.74} C_VEL
LIN {X 0,Y 94.384,Z 465.801,A -85,B 0,C 180,E1 -29790,E2 -29790} C_VEL
LIN {X 0,Y 85.221,Z 465.491,A -85,B 0,C 180,E1 -29798.286,E2 -29798.286} C_VEL
LIN {X 0,Y 80.208,Z 464.437,A -85,B 0,C 180,E1 -29805.466,E2 -29805.466} C_VEL
LIN {X 0,Y 76.765,Z 462.602,A -85,B 0,C 180,E1 -29813.728,E2 -29813.728} C_VEL
LIN {X 0,Y 75.418,Z 459.741,A -85,B 0,C 180,E1 -29823.004,E2 -29823.004} C_VEL
LIN {X 0,Y 75.938,Z 456.765,A -85,B 0,C 180,E1 -29830.379,E2 -29830.379} C_VEL
LIN {X 0,Y 78.346,Z 452.155,A -85,B 0,C 180,E1 -29839.043,E2 -29839.043} C_VEL
LIN {X 0,Y 80.087,Z 449.037,A -85,B 0,C 180,E1 -29844.265,E2 -29844.265} C_VEL
LIN {X 0,Y 81.332,Z 446.194,A -85,B 0,C 180,E1 -29848.775,E2 -29848.775} C_VEL
LIN {X 0,Y 81.588,Z 444.924,A -85,B 0,C 180,E1 -29851.383,E2 -29851.383} C_VEL
LIN {X 0,Y 81.151,Z 443.571,A -85,B 0,C 180,E1 -29855.44,E2 -29855.44} C_VEL
LIN {X 0,Y 80.198,Z 442.722,A -85,B 0,C 180,E1 -29859.595,E2 -29859.595} C_VEL
LIN {X 0,Y 78.491,Z 441.18,A -85,B 0,C 180,E1 -29871.436,E2 -29871.436} C_VEL
LIN {X 0,Y 79.675,Z 439.897,A -85,B 0,C 180,E1 -29880.003,E2 -29880.003} C_VEL
LIN {X 0,Y 79.007,Z 440.856,A -85,B 0,C 180,E1 -29885.106,E2 -29885.106} C_VEL
LIN {X 0,Y 78.361,Z 442.301,A -85,B 0,C 180,E1 -29890.336,E2 -29890.336} C_VEL
LIN {X 0,Y 77.098,Z 444.779,A -85,B 0,C 180,E1 -29895.874,E2 -29895.874} C_VEL
LIN {X 0,Y 76.528,Z 445.76,A -85,B 0,C 180,E1 -29897.63,E2 -29897.63} C_VEL
LIN {X 0,Y 73.42,Z 448.756,A -85,B 0,C 180,E1 -29901.046,E2 -29901.046} C_VEL
LIN {X 0,Y 72.049,Z 449.926,A -85,B 0,C 180,E1 -29902.078,E2 -29902.078} C_VEL
LIN {X 0,Y 62.991,Z 455.95,A -85,B 0,C 180,E1 -29906.803,E2 -29906.803} C_VEL
LIN {X 0,Y 54.454,Z 460.698,A -85,B 0,C 180,E1 -29912.976,E2 -29912.976} C_VEL
LIN {X 0,Y 46.756,Z 464.312,A -85,B 0,C 180,E1 -29921.275,E2 -29921.275} C_VEL
LIN {X 0,Y 42.262,Z 466.116,A -85,B 0,C 180,E1 -29928.304,E2 -29928.304} C_VEL
LIN {X 0,Y 35.978,Z 468.583,A -85,B 0,C 180,E1 -29947.003,E2 -29947.003} C_VEL
LIN {X 0,Y 34.48,Z 469.184,A -85,B 0,C 180,E1 -29958.239,E2 -29958.239} C_VEL
LIN {X 0,Y 34.241,Z 469.349,A -85,B 0,C 180,E1 -29970,E2 -29970} C_VEL
LIN {X 0,Y 34.473,Z 469.183,A -85,B 0,C 180,E1 -29981.763,E2 -29981.763} C_VEL
LIN {X 0,Y 35.974,Z 468.583,A -85,B 0,C 180,E1 -29992.999,E2 -29992.999} C_VEL
LIN {X 0,Y 42.262,Z 466.116,A -85,B 0,C 180,E1 -30011.696,E2 -30011.696} C_VEL
LIN {X 0,Y 49.207,Z 463.16,A -85,B 0,C 180,E1 -30021.77,E2 -30021.77} C_VEL
LIN {X 0,Y 57.255,Z 459.168,A -85,B 0,C 180,E1 -30029.231,E2 -30029.231} C_VEL
LIN {X 0,Y 66.264,Z 453.851,A -85,B 0,C 180,E1 -30035.04,E2 -30035.04} C_VEL
LIN {X 0,Y 72.043,Z 449.925,A -85,B 0,C 180,E1 -30037.933,E2 -30037.933} C_VEL
LIN {X 0,Y 74.68,Z 447.576,A -85,B 0,C 180,E1 -30040.233,E2 -30040.233} C_VEL
LIN {X 0,Y 76.486,Z 445.79,A -85,B 0,C 180,E1 -30042.364,E2 -30042.364} C_VEL
LIN {X 0,Y 77.842,Z 443.377,A -85,B 0,C 180,E1 -30046.952,E2 -30046.952} C_VEL
LIN {X 0,Y 78.469,Z 442.113,A -85,B 0,C 180,E1 -30050.132,E2 -30050.132} C_VEL
LIN {X 0,Y 79.003,Z 440.859,A -85,B 0,C 180,E1 -30054.894,E2 -30054.894} C_VEL
LIN {X 0,Y 79.693,Z 439.883,A -85,B 0,C 180,E1 -30059.997,E2 -30059.997} C_VEL
LIN {X 0,Y 78.397,Z 441.383,A -85,B 0,C 180,E1 -30069.562,E2 -30069.562} C_VEL
LIN {X 0,Y 77.794,Z 443.051,A -85,B 0,C 180,E1 -30075.722,E2 -30075.722} C_VEL
LIN {X 0,Y 77.56,Z 443.985,A -85,B 0,C 180,E1 -30078.487,E2 -30078.487} C_VEL
LIN {X 0,Y 76.603,Z 446.039,A -85,B 0,C 180,E1 -30083.443,E2 -30083.443} C_VEL
LIN {X 0,Y 75.71,Z 448.015,A -85,B 0,C 180,E1 -30087.651,E2 -30087.651} C_VEL
LIN {X 0,Y 74.523,Z 450.271,A -85,B 0,C 180,E1 -30091.924,E2 -30091.924} C_VEL
LIN {X 0,Y 72.093,Z 453.922,A -85,B 0,C 180,E1 -30098.75,E2 -30098.75} C_VEL
LIN {X 0,Y 69.175,Z 458.448,A -85,B 0,C 180,E1 -30108.671,E2 -30108.671} C_VEL
LIN {X 0,Y 68.597,Z 461.836,A -85,B 0,C 180,E1 -30119.185,E2 -30119.185} C_VEL
LIN {X 0,Y 69.589,Z 463.489,A -85,B 0,C 180,E1 -30126.173,E2 -30126.173} C_VEL
LIN {X 0,Y 75.348,Z 465.628,A -85,B 0,C 180,E1 -30139.249,E2 -30139.249} C_VEL
LIN {X 0,Y 79.772,Z 466.061,A -85,B 0,C 180,E1 -30144.946,E2 -30144.946} C_VEL
LIN {X 0,Y 85.174,Z 466.055,A -85,B 0,C 180,E1 -30150,E2 -30150} C_VEL
LIN {X 0,Y 77.92,Z 465.892,A -85,B 0,C 180,E1 -30157.211,E2 -30157.211} C_VEL
LIN {X 0,Y 71.951,Z 464.723,A -85,B 0,C 180,E1 -30167.04,E2 -30167.04} C_VEL
LIN {X 0,Y 69.475,Z 463.34,A -85,B 0,C 180,E1 -30174.443,E2 -30174.443} C_VEL
LIN {X 0,Y 68.467,Z 460.624,A -85,B 0,C 180,E1 -30184.802,E2 -30184.802} C_VEL
LIN {X 0,Y 69.882,Z 456.991,A -85,B 0,C 180,E1 -30194.748,E2 -30194.748} C_VEL
LIN {X 0,Y 72.754,Z 452.909,A -85,B 0,C 180,E1 -30203.08,E2 -30203.08} C_VEL
LIN {X 0,Y 74.899,Z 449.626,A -85,B 0,C 180,E1 -30209.367,E2 -30209.367} C_VEL
LIN {X 0,Y 75.693,Z 448.027,A -85,B 0,C 180,E1 -30212.342,E2 -30212.342} C_VEL
LIN {X 0,Y 77.012,Z 445.175,A -85,B 0,C 180,E1 -30218.594,E2 -30218.594} C_VEL
LIN {X 0,Y 77.563,Z 443.983,A -85,B 0,C 180,E1 -30221.513,E2 -30221.513} C_VEL
LIN {X 0,Y 78.333,Z 441.546,A -85,B 0,C 180,E1 -30229.666,E2 -30229.666} C_VEL
LIN {X 0,Y 78.491,Z 441.18,A -85,B 0,C 180,E1 -30231.436,E2 -30231.436} C_VEL
LIN {X 0,Y 78.187,Z 441.158,A -85,B 0,C 180,E1 -30234.275,E2 -30234.275} C_VEL
LIN {X 0,Y 77.184,Z 441.842,A -85,B 0,C 180,E1 -30237.056,E2 -30237.056} C_VEL
LIN {X 0,Y 72.909,Z 445.701,A -85,B 0,C 180,E1 -30246.669,E2 -30246.669} C_VEL
LIN {X 0,Y 71.867,Z 447.294,A -85,B 0,C 180,E1 -30252.065,E2 -30252.065} C_VEL
LIN {X 0,Y 71.18,Z 448.216,A -85,B 0,C 180,E1 -30254.291,E2 -30254.291} C_VEL
LIN {X 0,Y 69.533,Z 449.714,A -85,B 0,C 180,E1 -30256.218,E2 -30256.218} C_VEL
LIN {X 0,Y 68.059,Z 450.883,A -85,B 0,C 180,E1 -30257.218,E2 -30257.218} C_VEL
LIN {X 0,Y 57.02,Z 457.417,A -85,B 0,C 180,E1 -30262.421,E2 -30262.421} C_VEL
LIN {X 0,Y 47.988,Z 461.744,A -85,B 0,C 180,E1 -30268.513,E2 -30268.513} C_VEL
LIN {X 0,Y 42.387,Z 464.115,A -85,B 0,C 180,E1 -30274.002,E2 -30274.002} C_VEL
LIN {X 0,Y 37.238,Z 465.919,A -85,B 0,C 180,E1 -30280.981,E2 -30280.981} C_VEL
LIN {X 0,Y 29.54,Z 468.386,A -85,B 0,C 180,E1 -30301.586,E2 -30301.586} C_VEL
LIN {X 0,Y 27.549,Z 468.987,A -85,B 0,C 180,E1 -30315.22,E2 -30315.22} C_VEL
LIN {X 0,Y 27.127,Z 469.153,A -85,B 0,C 180,E1 -30330,E2 -30330} C_VEL
LIN {X 0,Y 27.542,Z 468.987,A -85,B 0,C 180,E1 -30344.784,E2 -30344.784} C_VEL
